METHOD MoveModulo 								: REFERENCE TO Tc2_MC2.ST_McOutputs
VAR_INPUT
	bExecute									: BOOL;
END_VAR
END_METHOD

METHOD MoveModulo2 								: REFERENCE TO Tc2_MC2.ST_McOutputs
VAR_INPUT
	bExecute									: BOOL;
END_VAR
END_METHOD

METHOD MoveModuloClear 							: BOOL
END_METHOD

METHOD MoveModuloClear2 						: BOOL
END_METHOD

METHOD MoveModuloCurrent 						: REFERENCE TO Tc2_MC2.ST_McOutputs
VAR_INPUT
	bExecute									: BOOL;
END_VAR
END_METHOD

METHOD MoveModuloCurrent2 						: REFERENCE TO Tc2_MC2.ST_McOutputs
VAR_INPUT
	bExecute									: BOOL;
END_VAR
END_METHOD

METHOD MoveModuloEx 							: BOOL
END_METHOD

METHOD MoveModuloEx2 							: BOOL
END_METHOD

METHOD MoveModuloNeg 							: REFERENCE TO Tc2_MC2.ST_McOutputs
VAR_INPUT
	bExecute									: BOOL;
END_VAR
END_METHOD

METHOD MoveModuloNeg2 							: REFERENCE TO Tc2_MC2.ST_McOutputs
VAR_INPUT
	bExecute									: BOOL;
END_VAR
END_METHOD

METHOD MoveModuloPos 							: REFERENCE TO Tc2_MC2.ST_McOutputs
VAR_INPUT
	bExecute									: BOOL;
END_VAR
END_METHOD

METHOD MoveModuloPos2 							: REFERENCE TO Tc2_MC2.ST_McOutputs
VAR_INPUT
	bExecute									: BOOL;
END_VAR
END_METHOD

METHOD MoveModuloShort 							: REFERENCE TO Tc2_MC2.ST_McOutputs
VAR_INPUT
	bExecute									: BOOL;
END_VAR
END_METHOD

METHOD MoveModuloShort2 						: REFERENCE TO Tc2_MC2.ST_McOutputs
VAR_INPUT
	bExecute									: BOOL;
END_VAR
END_METHOD

METHOD MoveRelative 							: REFERENCE TO Tc2_MC2.ST_McOutputs
VAR_INPUT
	bExecute									: BOOL;
END_VAR
END_METHOD

METHOD MoveRelative2 							: REFERENCE TO Tc2_MC2.ST_McOutputs
VAR_INPUT
	bExecute									: BOOL;
END_VAR
END_METHOD

METHOD MoveRelativeClear 						: BOOL
END_METHOD

METHOD MoveRelativeClear2 						: BOOL
END_METHOD

METHOD MoveRelativeEx 							: BOOL
END_METHOD

METHOD MoveRelativeEx2 							: BOOL
END_METHOD

METHOD MoveVelocity 							: REFERENCE TO Tc2_MC2.ST_McOutputs
VAR_INPUT
	bExecute									: BOOL;
END_VAR
END_METHOD

METHOD MoveVelocity2 							: REFERENCE TO Tc2_MC2.ST_McOutputs
VAR_INPUT
	bExecute									: BOOL;
END_VAR
END_METHOD

METHOD MoveVelocityClear 						: BOOL
END_METHOD

METHOD MoveVelocityClear2 						: BOOL
END_METHOD

METHOD MoveVelocityEx 							: BOOL
END_METHOD

METHOD MoveVelocityEx2 							: BOOL
END_METHOD

PROPERTY nErrorId 								: UDINT
GET
END_GET
END_PROPERTY

PROPERTY pAbsolute 								: REFERENCE TO Tc2_MC2.ST_McOutputs
GET
END_GET
SET
END_SET
END_PROPERTY

PROPERTY pAbsolute2 							: REFERENCE TO Tc2_MC2.ST_McOutputs
GET
END_GET
SET
END_SET
END_PROPERTY

PROPERTY pEStop 								: REFERENCE TO Tc2_MC2.ST_McOutputs
GET
END_GET
SET
END_SET
END_PROPERTY

PROPERTY pGear 									: REFERENCE TO Tc2_MC2.ST_McOutputs
GET
END_GET
SET
END_SET
END_PROPERTY

PROPERTY pHalt 									: REFERENCE TO Tc2_MC2.ST_McOutputs
GET
END_GET
SET
END_SET
END_PROPERTY

PROPERTY pHome 									: REFERENCE TO Tc2_MC2.ST_McOutputs
GET
END_GET
SET
END_SET
END_PROPERTY

PROPERTY pJog 									: REFERENCE TO Tc2_MC2.ST_McOutputs
GET
END_GET
SET
END_SET
END_PROPERTY

PROPERTY pLimitSwitch 							: REFERENCE TO Tc2_MC2.ST_McOutputs
GET
END_GET
SET
END_SET
END_PROPERTY

PROPERTY pModulo 								: REFERENCE TO Tc2_MC2.ST_McOutputs
GET
END_GET
SET
END_SET
END_PROPERTY

PROPERTY pModulo2 								: REFERENCE TO Tc2_MC2.ST_McOutputs
GET
END_GET
SET
END_SET
END_PROPERTY

PROPERTY pOut 									: REFERENCE TO Tc2_MC2.ST_McOutputs
GET
END_GET
SET
END_SET
END_PROPERTY

METHOD Power 									: REFERENCE TO Tc2_MC2.ST_McOutputs
END_METHOD

PROPERTY pPower 								: REFERENCE TO Tc2_MC2.ST_McOutputs
GET
END_GET
SET
END_SET
END_PROPERTY

PROPERTY pRelative 								: REFERENCE TO Tc2_MC2.ST_McOutputs
GET
END_GET
SET
END_SET
END_PROPERTY

PROPERTY pRelative2 							: REFERENCE TO Tc2_MC2.ST_McOutputs
GET
END_GET
SET
END_SET
END_PROPERTY

PROPERTY pReset 								: REFERENCE TO Tc2_MC2.ST_McOutputs
GET
END_GET
SET
END_SET
END_PROPERTY

PROPERTY pSetPos 								: REFERENCE TO Tc2_MC2.ST_McOutputs
GET
END_GET
SET
END_SET
END_PROPERTY

PROPERTY pStop 									: REFERENCE TO Tc2_MC2.ST_McOutputs
GET
END_GET
SET
END_SET
END_PROPERTY

PROPERTY pVelocity 								: REFERENCE TO Tc2_MC2.ST_McOutputs
GET
END_GET
SET
END_SET
END_PROPERTY

PROPERTY pVelocity2 							: REFERENCE TO Tc2_MC2.ST_McOutputs
GET
END_GET
SET
END_SET
END_PROPERTY

METHOD Reset 									: REFERENCE TO Tc2_MC2.ST_McOutputs
VAR_INPUT
	bExecute									: BOOL;
END_VAR
END_METHOD

METHOD ResetClear 								: BOOL
END_METHOD

METHOD ResetEx 									: BOOL
END_METHOD

METHOD SetPos 									: REFERENCE TO Tc2_MC2.ST_McOutputs
VAR_INPUT
	bExecute									: BOOL;
	bMode										: BOOL;	// RELATIVE=True, ABSOLUTE=False (Default)
	stOptions									: ST_SetPositionOptions;
END_VAR
END_METHOD

METHOD SetPosClear 								: BOOL
END_METHOD

METHOD SetPosEx 								: BOOL
VAR_INPUT
	bMode										: BOOL;	// RELATIVE=True, ABSOLUTE=False (Default)
	stOptions									: ST_SetPositionOptions;
END_VAR
END_METHOD

METHOD Stop 									: REFERENCE TO Tc2_MC2.ST_McOutputs
VAR_INPUT
	bExecute									: BOOL;
END_VAR
END_METHOD

METHOD StopClear 								: BOOL
END_METHOD

METHOD StopEx 									: BOOL
END_METHOD

END_INTERFACE

// ---- POUs/MAIN.TcPOU
PROGRAM MAIN
VAR_INPUT
	bWeighingFormDone											: BOOL;
	IbTwoPhasesFormSensorBetweenDispencers			AT %I*		: BOOL;		// Wejście czujnika pomiedzy dozownikami do przesuwania formatek
	IbFormCheckFormSensor 							AT %I*		: BOOL;		// Wejście wykrycia formatek przed szlabanem
	IbBottleInFormCheckBottleSensor 				AT %I*		: BOOL;		// Wejscie wykrycia butelki przed szlabane
	IbFourthFormCheckFormSensor						AT %I*		: BOOL;	
	IbSecondFormCheckFormSensor						AT %I*		: BOOL;	

	(*CapSorterDrag*)
	IbCapSorterFourthFormCheckFormSensor						: BOOL;
	IbCapSorterBeforeFourthFormCheckFormSensor					: BOOL;
	IbCapSorterAfterFormSensor 									: BOOL;
	IbCapSorterAfterFormSensor2 								: BOOL;		
	IbCapSorterAfterFormSensor3 					AT %I*		: BOOL;			
	IbCapSorterFirstFormCheckFormSensor 						: BOOL;		
	IbLidSealerFirstFormSensor						AT %I*:BOOL;			// Czujnik obecności 2-ej formatki przygrzewacze platynek
	IbLidSealerSecondFormSensor 								: BOOL;		// Czujnik obecności 2-ej formatki przygrzewacze platynek
	IbLidSealerAfterSensor 										: BOOL;		// Czujnik obecności formatek przygrzewacze platynek wyjazd
	IbBlowBeforeGripperScrewerSensor							: BOOL;
	IbLidFeederThirdFormSensor 							AT %I*  : BOOL;		// Czujnik obecności formatki trzecia formatka 
	IbLidFeederAfterSensor 								AT %I*  : BOOL;		// Czujnik obecności formatki wyjazd	
END_VAR
VAR
	fbReasonBadPackage1											: FB_ReasonBadPackage;
	fbReasonBadPackage2											: FB_ReasonBadPackage;
	fb2ReasonBadPackageWithID									: FB_2ReasonBadPackageWithID;	
	
	fbMRBottleFeederPackageState								: FB_MoveRegister;
	fbMRBeforeDispencersPackageStateNew							: FB_MoveRegister;
	fbMRDispencerPackageState									: FB_MoveRegister4;//Sprzed dozowników na dozowniki
	fbMRAfterDispencerPackageState								: FB_MoveRegister4;//z dozowników za dozowniki
	fbMRWeightPackageState										: FB_MoveRegister; // zza dozowników na wage
	fbMRWeight2PhasePackageState								: FB_MoveRegister; // zza dozowników na wage 2 fazy
	fbMRAfterWeightPackageState									: FB_MoveRegister; // z wagi na transporter
	fbMRBEforeScrewer2PackageState								: FB_MoveRegisterSortAndMove;
	fbMRBeforeScrewerPackageState								: FB_MoveRegisterCapControl; // Przed zakręcarkami

	fbMRCorrectCapPackageState									: FB_MoveRegister; // zza zakręcarek na kontrole zakreceniea
	
// Dodatkowe przesuwanie rejestrów 
	
	fbMRBeforeDispencer34PackageState							: FB_MoveRegister;
	fbMRAfterDispencer34PackageState							: FB_MoveRegister4;
	fbMRDispencer34PackageState									: FB_MoveRegister4;
	fbMRBetweenDispencerPackageState							: FB_MoveRegister; 
	fbMRAfterDispencer12PackageState							: FB_MoveRegister4;
	fbMRDispencer12PackageState									: FB_MoveRegister4;

	
	
// LidFeeder
	fbMRBeforeLidFeeder2PackageState							: FB_MoveRegisterSortAndMoveLF;
	fbMRAfterWeightPackageStateLF								: FB_MoveRegisterLF; // z wagi na transporter
	fbIbLidFeederThirdFormSensor								: FB_InputFilter_V2;
	ftfbIbLidFeederThirdFormSensor								: F_TRIG;
	bMRBeforeLidFeeder2Block									: BOOL;
	rtfbIbLidFeederThirdFormSensor								: R_TRIG;
	ftbMRBeforeLidFeeder2Block									: F_TRIG;
	tofftbMRBeforeLidFeeder2Block								: TOF;	
	bMRLidFeederFormInCap										: BOOL;
// LidFeederDrag
	rtfbLidFeederDrag											: R_TRIG;

//AfterLidFeeder
	fbMRAfterLidFeederPackageState								: FB_MoveRegister; // zza zakręcarek na kontrole zakreceniea
	ftfbIbLidFeederAfterSensor									: F_TRIG;
	rtfbIbLidFeederAfterSensor									: R_TRIG;
	fbIbLidFeederAfterSensor									: FB_InputFilter;

//LidSealer
	rtfbLidSealerDrag											: R_TRIG;
	
	
	fbIbFirstFormCheckFormSensor								: FB_InputFilter_v2;
	fbIbSecondFormCheckFormSensor								: FB_InputFilter_v2;
	fbFilteredFormsSensorGate 									: FB_InputFilter;
	fbIbCapCorrectCheckFormSensor								: FB_InputFilter;
	fbIbScrewerThirdFormCheckFormSensor							: FB_InputFilter;
	fbIbCapPuttedCheckFormSensor								: FB_InputFilter;
	fbIbCapPuttedCheckFormSensorv2								: FB_InputFilter_v2;
	fbIbWeight1FormSensor										: FB_InputFilter_v2;
	fbIbWeight4FormSensor										: FB_InputFilter_v2;
	fbIbCapPuttedCheckFormSensorAfterStart						: FB_InputFilter;
	fbIbScrewerThirdFormCheckFormSensorAfterStart				: FB_InputFilter;
	
	fbIbBottleFeederFormPresent									: FB_InputFilter;
	
	
	
	
	bRFIDArrayClear												: BOOL;
	bDeletebBottleTransferedToExit								: BOOL;
	bNewRFIDSaved												: BOOL;
	
	bWeighingFormDoneDialog										: BOOL;
	bWeighingFormReset											: BOOL;

	bNewRFIDSaved1												: BOOL;
	bNewRFIDSaved2												: BOOL;
	bNewRFIDSaved3												: BOOL;
	bNewRFIDSaved4												: BOOL;
	//Sygnały obecnosci formatek przed dozownikami

	
	
	
	bKeepTryingMove1,bKeepTryingMove2,bKeepTryingMove3,bKeepTryingMove4  		: BOOL;
	bKeepTryingMove5,bKeepTryingMove6,bKeepTryingMove7,bKeepTryingMove8	 		: BOOL;
	bKeepTryingMove9,bKeepTryingMove10,bKeepTryingMove11,bKeepTryingMove12	 	: BOOL;
	bKeepTryingMove13,bKeepTryingMove14,bKeepTryingMove15	 					: BOOL;
	bKeepTryingMove17,bKeepTryingMove18,bKeepTryingMove19,bKeepTryingMove20	 	: BOOL;
	bKeepTryingMove799,bKeepTryingMove798,bKeepTryingMove797,bKeepTryingMove796	 : BOOL;
	
	
	bMRFormExitGate1											: BOOL;
	bMRFormDispencer											: BOOL;
	bMRFormExitDispencer										: BOOL;
	bMRFormExitWeight											: BOOL;
	bMRFormInCap												: BOOL;
	bMRCapCorrect												: BOOL;
// Dodatkowe zmienne dla dwufazy
	bMRFormDispencer12											: BOOL;
	bMRFormDispencer34											: BOOL;
	bMRFormExitDispencer12										: BOOL;
	bMRFormExitDispencer34										: BOOL;
	bMRFormBetweenDispencer										: BOOL;
	

	bResetHistory												: BOOL;
	bSimulationForLoop											: BOOL;
	bTestBrakePoint												: BOOL;
	bMRBeforeScrewer2Block										: BOOL;
	bTemp														: BOOL;
	bTrendIbThirdFormCheckFormSensor							: BOOL;
	bTrendFilteredIbThirdFormCheckFormSensor					: BOOL;

	bRFIDSBeforeScrewerWriteToRegister							: BOOL;
	
	
	nFormCounter												: INT;
	nCheckRobotDone												: INT;
	is															: INT;
	iCountSimulation											: INT;
	ir1															: INT;
	ir2															: INT;
	ir3															: INT;
	ir4															: INT;
	ir5															: INT;
	id															: INT;
	ia															: INT;
	iw															: INT;
	iftfbIbCapPuttedCheckFormSensor								: INT;
	iBadPackage1ReasonCount1									: INT;
	iBadPackage1ReasonCount2									: INT;
	iBadPackage1ReasonCount3									: INT;
	iBadPackage2ReasonCount1									: INT;
	iBadPackage2ReasonCount2									: INT;
	iBadPackage2ReasonCount3									: INT;
	ifbIbCapPuttedCheckFormSensorAfterStart						: INT;
	ifbIbScrewerThirdFormCheckFormSensorAfterStart				: INT;
	irtTimerRFIDScrewersWarning									: INT;
	iRFIDSBeforeScrewerWriteToRegister							: INT;
	
	i															: UINT;
	nr1															: UINT;
	nr2															: UINT;
	nr3															: UINT;
	nr4															: UINT;
	nr5															: UINT;	
	nr6															: UINT;	
	nr7															: UINT;	
	nr8															: UINT;	
	
	nSimulationCardNumber										: ULINT;

	sBadPackage1Reason1											: STRING;
	sBadPackage1Reason2											: STRING;
	sBadPackage1Reason3											: STRING;
	sBadPackage2Reason1											: STRING;
	sBadPackage2Reason2											: STRING;
	sBadPackage2Reason3											: STRING;
	
	// RFID
	rtReadedCardDispencer										: R_TRIG;
	rtReadedCardBeforeScrewers									: R_TRIG;
	rtReadedCardAfterScrewers									: R_TRIG;	
	rtReadedCardAfterDispencers									: R_TRIG;
	rtReadedCardAfterDispencers2Phase							: R_TRIG;
	rtReadedCardLidFeeder										: R_TRIG;
	rtReadedCardLidSealer										: R_TRIG;
	rtReadedCardCapSorter										: R_TRIG;	
	rtReadedCardRobotTransfer									: R_TRIG;
	fbrtReadedCardRobotTransfer									: FB_InputFilter_v2;
	fbrtReadedCardAfterScrewers									: FB_InputFilter_v2;
	rtWeighingForm												: R_TRIG;
	rtWeightingDone												: R_TRIG;
	rtBeforeGateDispencerStateNotPresent						: R_TRIG;
	rtBeforeGateDispencerFormPresent							: R_TRIG;
	rtSimulationSetRegisters									: R_TRIG;
	ftfbIbFirstFormCheckFormSensor								: F_TRIG;
	rtfbIbFirstFormCheckFormSensor								: R_TRIG;

	rtfbIbSecondFormCheckFormSensor								: R_TRIG;
	ftfbIbSecondFormCheckFormSensor								: F_TRIG;
	ftfbIbCapCorrectCheckFormSensor								: F_TRIG;
	rtfbIbCapCorrectCheckFormSensor								: R_TRIG;	
	rtfbFormsDragingPneumaticStationDragging					: R_TRIG;
	ftfbIbScrewerThirdFormCheckFormSensor						: F_TRIG;
	ftfbIbCapPuttedCheckFormSensor								: F_TRIG;
	ftfbIbWeight1FormSensor										: F_TRIG;
	ftIbWeight4FormSensor										: F_TRIG;
	ftbMRBeforeScrewer2Block									: F_TRIG;
	rttonDelayAfterStart										: R_TRIG;
	rtfbIbScrewerThirdFormCheckFormSensor						: R_TRIG;
	rtTimerRFIDScrewersWarning									: R_TRIG;
	
	diRFIDWeightingFormNumber									:DINT;
	tonAfter1stweight											:TON;
	bWeightEnd													:BOOL;
	
	tonWeighingForm												: TON;
	tonFourthFormBeforeDispencerCheck							: TON;
	tofCycleExecute												: TOF;
	tonFormBeforeDispenscerCheck								: TON;
	tonDispencerRepair1											: TON;
	TimerRFIDWeightWarning										: TON;
	tonRobotPackageStatebBottleTransferedToLabeler				: TON;
	tonRobotPackageStatebBottleTransferedToLabeler2				: TON;
	TimerRFIDDispencersWarning									: TON;
	TimerRFIDDispencers2PhaseWarning							: TON;
	TimerRFIDScrewersWarning									: TON;
	TimerRFIDRobotWarning										: TON;
	tofftbMRBeforeScrewer2Block									: TOF;
	tonAfterDispencersRepair									: TON;
	tonAfterDispencersRepair1B									: TON;
	tonAfterDispencersRepair2									: TON;	
	tonAfterDispencersRepair3									: TON;	
	tonAfterDispencersRepair4									: TON;	
	tonRepairLidFeeder1											: TON;		
	tonRepairLidFeeder2											: TON;	
	tonRepairLidFeeder3											: TON;	
	tonRepairLidFeeder4											: TON;	
		
	// dodatkowe zmienne przy dwufazie
	fbIbWeight5FormSensor										: FB_InputFilter_v2;
	fbIbWeight6FormSensor										: FB_InputFilter_v2;

	ftfbIbWeight5FormSensor										: F_TRIG;
	ftIbWeight6FormSensor										: F_TRIG;
	
	//
	
	
	
	rtWeightingDone2Phase										: R_TRIG;
	ftfbIbBottleFeederFormPresent								: F_TRIG;
	
	rtibBottleFeederrFormPresent									: R_TRIG;
	bBitTestOn: BOOL;
	tonFormBeforeDispenscer2PhaseCheck							: TON;
	bTestCounterDispencer										: INT;
	tonRobotPackageStateFormsTooLong							: TON;
	tonRobotPackageState1FormsTooLong							: TON;
	tonRobotPackageState2FormsTooLong							: TON;
	END															: INT;
	ftFormSensorBetweenDispencer								: F_TRIG;
	
	fbIbFormSensorBetweenDispencer								: FB_InputFilter_v2;
	
	tonUnderScrewerFormStuck1									: TON;
	tonUnderScrewerFormStuck2									: TON;
	tonAfterScrewerFormStuck1									: TON;
	iRFIDClearNr1AfterRobotCount								: INT;
	iRFIDClearNr2AfterRobotCount								: INT;
	rtiBottleTransferCase2										: R_TRIG;
	tonAfterDispencer12Repair									: TON;
	rttonAfterDispencer12Repair									: R_TRIG;
	
	tonAfterDispencer1234Repair									: TON;
	tonAfterDispencer1234Repair2								: TON;
	
	tonWeightRepair1											: TON;
	tonWeightRepair2											: TON;	
	rttonAfterDispencer1234Repair								: R_TRIG;
	tonFourhtFormBeforeDispencer34								: TON;
	rttonFourtFormBeforeDispencer34Repair						: R_TRIG;
	rtFormSensorBetweenDispencer								: R_TRIG;
	fbIbCapCorrectCheckAfterScrewerFormSensor					: FB_InputFilter;
	ftfbIbCapCorrectCheckAfterScrewerFormSensor					: F_TRIG;
	
	rtTimerRFIDDispencerWarning: R_TRIG;
	irtTimerRFIDDispencerWarning: INT;
	tWeightTime: TIME;
	
	(*RFID*)
	bRFIDRepairAddNumber								: BOOL;
	iRFIDRepairAddNumber								: INT;
	nRFIDRepairOrderFirstNumber							: ULINT;
	AbRFIDRepairOrderTemp								: ULINT;
	nRFIDRepairToRotate									: ULINT;
	nRFIDRepairFormToRotateCount						: ULINT;
	bRFIDRepairChanged									: BOOL;
	iWeightPackageState12nCardNumberChangeCounter		: INT;
	iWeightPackageState13nCardNumberChangeCounter		: INT;


	
	bRFIDRepairReset: BOOL;
	rtRFIDRepairAddNumber: R_TRIG;
	nBeforeGatePackageState1nCardNumber: ULINT;
	ftRFIDRepairAddNumber: F_TRIG;
	rtRFIDRepairToRotate: R_TRIG;
	nRFIDRepairToRotateBefore: ULINT;
	fbRFIDRepairFilteredFormsSensorGate: FB_InputFilter;
	iRFIDRepairCount1: INT;
	iRFIDRepairCount2: INT;
	iRFIDRepairCount3: INT;
	iRFIDRepairCount4: INT;
	iRFIDRepairCount5: INT;
	bRFIDRepairOrderFirstNumberSaved: BOOL;
	iRFIDRepairCount6: INT;
	iRFIDRepairCount7: INT;
	iWeightPackageState43nCardNumberChangeCounter: INT;
	iWeightPackageState41nCardNumberChangeCounter: INT;
	iWeightPackageState21nCardNumberChangeCounter: INT;
	iWeightPackageState32nCardNumberChangeCounter: INT;
	iWeightPackageState31nCardNumberChangeCounter: INT;
	iUnderScrewerPackageState21nCardNumberChangeCounter: INT;
	iRFIDRepairCount8: INT;
	iRFIDRepairNumberOfForms: INT;
	iUnderScrewerPackageState12nCardNumberChangeCounter: INT;

	rtbBottleDragingStationRun: R_TRIG;
	rtDispencerDragStation: R_TRIG;

	rttonUnderScrewerFormStuck1: R_TRIG;
	rttonRobotPackageStatebBottleTransferedToLabeler: R_TRIG;
	rttonRobotPackageStatebBottleTransferedToLabeler2: R_TRIG;
	rttonRobotPackageState1FormsTooLong: R_TRIG;
	rttonRobotPackageState2FormsTooLong: R_TRIG;
	rteUnderScrewerPackageStateCheck: R_TRIG;
	rteUnderScrewerPackageStateCheck2: R_TRIG;
	iUnderScrewerPackageStateCheckCounter: INT;
	iUnderScrewerPackageStateCheckCounter2: INT;
	tonDispencer34DosingAborted: TON;
	rttonDispencer34DosingAborted: R_TRIG;
	
	tonFormatSensorOn	:	ton;
	tonFormatSensorOff	:	ton;
	bFormatSensor		:	BOOL;

	tonBottleSensorOn	:	ton;
	tonBottleSensorOff	:	ton;
	bBottleSensor		:	BOOL;
	

	
	
	tonIbCapSorterAfterFormSensor						: TON;
	fbMRAfterCapSorterPackageState						: FB_MoveRegister4; // Z sortera za sorter
	fbMRCapSorterPackageState							: FB_MoveRegister4; // Sprzed sortera na sorter
	fbMRBeforeCapSorterPackageState						: FB_MoveRegister;
	fbFilteredCapSorterFormsSensorGate 					: FB_InputFilter;
	ftfbFilteredCapSorterFormsSensorGate				: F_TRIG;
	tonFormBeforeCapSorterCheck							: TON;
	
	
	iAfterDispencersFormCounter: INT;
	itonFormBeforeCapSorterCheck: INT;
	bResetAntyErrorCounters: BOOL;
	lrAnRFIDWeightShowAverage: LREAL;
	iAnRFIDWeightShowAverageCount: INT;
	bRFIDWeightShowAverageError: BOOL;	
	ii: UINT;
	

	
	iLFTest1: INT;
	j: INT;
	iTestCCC1: INT;
	iTestCCC2: INT;
	
	(*ROPP*)
	rtReadedCardBeforeROPP				: R_TRIG;
	rtReadedCardAfterROPP				: R_TRIG;
	iropp1, iropp2						: INT;
	bRFIDSBeforeROPPWriteToRegister		: BOOL;
	iRFIDSBeforeROPPWriteToRegister		: INT;
	rtfbROPPDrag						: R_TRIG;
	bMRBeforeROPP2Block					: BOOL;
	ftbMRBeforeROPP2Block 				: F_TRIG;
	tofftbMRBeforeROPP2Block			: TOF;
	fbMRBEforeROPP2PackageState			: FB_MoveRegisterSortAndMoveROPP;
	bKeepTryingMoveROPP1					: BOOL;	
	bROPPMR								: BOOL;	
	fbMRBeforeROPPPackageState			: FB_MoveRegisterROPPCapControl; 
	tonRepairROPP1						: TON;		
	tonRepairROPP2						: TON;	
	tonRepairROPP3						: TON;	
	tonRepairROPP4						: TON;		
	bKeepTryingMoveROPP2				: BOOL;
	iPodglad:UINT;
	
	fbShutdown_UBL :NT_Shutdown;
	fbShutdown_UCF :NT_Shutdown;
	fbShutdown_UBF :NT_Shutdown;
	
	 fbRenew : FB_AutoTrialRenew_ADS;
     bExpired : BOOL := FALSE;
	 btestlicense	:bool:=false;
END_VAR

TcMcGlobal.NCPORT_TCMC_RESET := 501; // Przeciw bluescreen'om

VIS.sType				:=	'UL50-0125';
VIS.sSerialNumber		:=	'UL50-0125';
VIS.rProgramVersion		:=	0.2; (*XD*)
VIS.rLastTimeChanges	:=	20252810;


//Resetowanie przeważania
IF bWeighingFormReset THEN
	
	FOR i := 1 TO 100 DO
		VIS.AnRFIDCardNumberShow[i]								:= 0;
		VIS.AnRFIDWeightShow[i]									:= 0;
	END_FOR
	
	bWeighingFormReset 											:= FALSE;
	bWeighingFormDone 											:= FALSE;
	bWeighingFormDoneDialog 									:= FALSE;
	iRFIDRepairCount1	:=0;
	iRFIDRepairCount2	:=0;
	iRFIDRepairCount3	:=0;
	iRFIDRepairCount4	:=0;
END_IF

aInFormatSensorFilter();

aWizard();
P00_SystemDiagnostics();
a0RemoteControl();
aAntyError();
aAntyErrorLidFeeder();
//aAntyErrorROPP();
aBadPackage();
aCycleLogicHMI();
aStatistics();
aSimulation();

//aRFIDRepairSignals();
//MAIN.aRFIDRepairReset();
//bRFIDChecker:=TRUE; 
bRFIDChecker:=FALSE;

IF bRFIDChecker	THEN
	MAIN.aRFIDRepairOrderCreate();
	MAIN.aRFIDRepairOrderSearch();
	MAIN.aRFIDRepairStatistic();
END_IF	

P00_Communication();
P00_PackML();			
P00_Alarms();
P00_Basic();
P00_Counters();
P00_Persistent();
P00_OEE();
P00_PneumaticValves();
P00_ReadRFIDCard();
P00_Recipes();
P00_Signalization();
P00_Visualization();
P01_TwoPhasesBarriers();
P01_BottleFeeder();
P01_PucksInserter();
P01_BottleSorter();
P01_Gates();
P02_BottlePusher();
P02_Dispencers();
P02_DispencersCharts();
P05_WeightCorrection();
//P05_Weight();
P06_LidFeeder();
//P06_WickFeeder();
P06_LidPuttedCheck();
P07_CapPusher();
P06_LidSealer();
P07_ROPP();
P08_CapFeeder();
P08_CapSorter();
P09_CapPuttedCheck();
P10_GripperScrewer();
P11_CapCorrectCheck();
P11_RollerScrewer();
P13_BottleTransfer();
P13_BottleTransferAfterDrag();
P14_BadBottleConyevor();
P15_FormTransporters();
P16_LabelMachine();
P17_TurnTables();
P20_ExhaustFan();
//P030_Recipes();
P010_AlarmsWarningsInfosLogs();
P020_RtcEffectivityOEE();
P009_ReadSavePersistent();
P_AdsLicenseServer();
P200_CapPreScrewer();

tofCycleExecute(IN:=	(P00_PackML.fbPMLAuto.ePMLState = E_PMLState.ePMLState_STARTING) OR (P00_PackML.fbPMLAuto.ePMLState = E_PMLState.ePMLState_EXECUTE) OR 
						(P00_PackML.fbPMLAuto.ePMLState = E_PMLState.ePMLState_STOPPING) OR (P00_PackML.fbPMLAuto.ePMLState = E_PMLState.ePMLState_ABORTING),PT:=T#2S);

IF  tofCycleExecute.Q THEN
	
	IF bDosingTwoPhases THEN
		MAIN.aCycleRegister2Phase();
	ELSE
		IF bLidFeederEnable OR bWickFeederEnable THEN
			MAIN.aCycleRegister1PhaseLidFeederOrWick();
		ELSE
			MAIN.aCycleRegister1Phase();
		END_IF
	END_IF
	
END_IF

aRFIDWarnings();


fbShutdown_UBL(
	NETID:= '192.168.40.180.1.1',
	DELAY:= 10,
	START:=vis.bOffPLC ,
	TMOUT:= ,
	BUSY=> ,
	ERR=> ,
	ERRID=> );
	
//fbShutdown_UCF(
//	NETID:= '192.168.40.155.1.1',
//	DELAY:= 10,
//	START:=vis.bOffPLC ,
//	TMOUT:= ,
//	BUSY=> ,
//	ERR=> ,
//	ERRID=> );	
//	
//fbShutdown_UBF(
//	NETID:= '192.168.40.151.1.1',
//	DELAY:= 10,
//	START:=vis.bOffPLC ,
//	TMOUT:= ,
//	BUSY=> ,
//	ERR=> ,
//	ERRID=> );

IF btestlicense THEN
    bExpired := TRUE;
END_IF
fbRenew(
    bExpired := bExpired,
    sProductId := 'TC1220',
    sAdsServerNetId := '192.168.40.180.1.1',    // AMS Net ID PLC z serwerem ADS
    nAdsServerPort := 851
);

// Nowa "licencja"
fbRenew.sLicenseOut;

ACTION a0RemoteControl:
(*
Nazwa:			a0RemoteControl
Opis:			Ulatwienie obsługi maszyny bez wizki
Wersja:			v0.1
Data:			2023-03-13
Autor:			DP
Urzadzenia:		
Konfiguracja:	
Info:
-


*)
{warning 'Dorobić błędy Undervoltage'}
VIS.bChooseRecipe ; P00_PackML.iChooseRecipe;
VIS.bRecipeLoading;P00_PackML.fbbRecipeLoading.bOut;

IbCycleStopButton;
IbCycleStartButton; 

VIS.bServiceMode;
VIS.bAllowStart ;
VIS.bSimulation;
VIS.bWeighingForm;

VIS.lrDispencersLifterReadyPositionShow;
VIS.lrDispencer1LifterStartDosePositionShow;
VIS.lrDispencer1LifterStopDosePositionShow;

VIS.bBottleTransferAllFormsToLabeler;
VIS.bBottleTransferAllFormsToExit;
VIS.iBottleTransferSpeedShow;	

stBottleSorterRead.ePackMLMode;
stBottleSorterRead.ePackMLAutoState; 
bBottleSorterDisable;

stCapSorterRead.ePackMLMode;
stCapSorterRead.ePackMLAutoState; 
bCapSorterDisable;
VIS.bCapPuttedCheckIgnoreErrors;

VIS.bResetErrorVisuCmd;
VIS.bErrorOccure;							
VIS.sStationInError;	
VIS.udiStationInError;			
VIS.udiStationErrorCode;			
VIS.sStationErrorDescription;	
VIS.sStationErrorDescription2;	

bHomingDialog;
VIS.bDialogBoxText;
VIS.bDialogBoxAck;

VIS.lrDispencer1DoseVolumeCV					;				// Doza 1 [ml]
VIS.lrDispencer2DoseVolumeCV					;				// Doza 2 [ml]
VIS.lrDispencer3DoseVolumeCV					;				// Doza 3 [ml]	
VIS.lrDispencer4DoseVolumeCV					;				// Doza 4 [ml]	
VIS.lrDispencer1WeightMeasured					;				// Waga z dozownika 1 [g]	
VIS.lrDispencer2WeightMeasured					;				// Waga z dozownika 2 [g]		
VIS.lrDispencer3WeightMeasured					;				// Waga z dozownika 3 [g]	
VIS.lrDispencer4WeightMeasured					;				// Waga z dozownika 4 [g]	
VIS.bDispencer1WeightMeasured					;				// [H] Waga zmierzona z dozownika nr 1	
VIS.bDispencer2WeightMeasured					;				// [H] Waga zmierzona z dozownika nr 2
VIS.bDispencer3WeightMeasured					;				// [H] Waga zmierzona z dozownika nr 3
VIS.bDispencer4WeightMeasured					;				// [H] Waga zmierzona z dozownika nr 4



iRepairFourthFormBeforeDispencerCounter;	// 1A - Ustawianie 4 formatki(*****************Autonaprawa przed dozownikami	*****************)
iRepairBeforeDispencer34Counter;			// 1B (2faza) - Autonaprawa 2 formatki przed dozowikiem 34
iCounterDispencer34DosingAborted;			// 1C (2faza) - Autonaprawa jak jest butelka a niewydozowało
iRepairFormBeforeDispenscerCounter;			// 1D - Ustawianie jak nie ma dwufazy - Ustawianie 1 2 3 4 formatki
iRepairFormBeforeDispenscer2PhaseCounter;	// 1E (2faza) - ustawianie jak jest dwufaza - Ustawianie 1 2  formatki
itonAfterDispencersRepair;					// 1 - Kasowanie rejestrow jezeli nie ma nic na czujnikach (******************Autonaprawa za dozownikami*************************)
itonAfterDispencersRepair2;					// 2 - Kasowanie rejestrow jezeli nei ma nic na czujnikach----------------
itonAfterDispencersRepair3;					// 3 - Kasowanie rejestrow jezeli nei ma nic na czujnikach --------------
itonAfterDispencersRepair4;					// 4 -  Kasowanie rejestrow jezeli nei ma nic na czujnikach-------------
iRepairAfterDispencerCounter;				// 4 - Kssowanie za 1 i 2 dozownikiem jak dwufaza -----------------------
iRepairBeforeDispencer12Counter;			// 5 - Dodawanie formatek przed 12 jak stoją za 34 ---------------------
iRepairBeforeDispencer12Counter2;
itonFormBeforeCapSorterCheck;				// 1A - Ustawianie 1 2 3 4 formatki(*****Autonaprawa pod sorterem nasadek**********)
iScrewerFormStuck;							// 1A - (****** Autonaprawa pod zakręcarkami*********)
iScrewerFormStuck2;							// 1B - jezeli nie odczyta przed zakrecarkami
iScrewerFormStuck3;							// 1S - jezeli nie ma za zakrecarka
iRobotRepairPackageForm1Counter;			// Jak jest przeniesiona na etykieciarke(*****Autonaprawa pod robotem**********)
iRobotRepairPackageForm2Counter;
itonRobotBottleTransferedToLabelerRepair;
itonRobotBottleTransferedToLabeler2Repair;
END_ACTION

ACTION a2RFID:
(*
Nazwa:			aRFID
Opis:			Zapisywanie RFID
Wersja:			v0.5
Data:			2024-12-02
Autor:			DP
Urzadzenia:		
Konfiguracja:	
Zmiany:
Info:
- zapis RFID do struktury
- text
*)

(*********************Wywoływane w aCycleLogic************************)

(*******************************)
(***CZUJNIK PRZED DOZOWNIKAMI***)

//Jeżeli wykryło kartę 
rtReadedCardDispencer(CLK:=P00_ReadRFIDCard.bReadedCardDispencer,Q=>);
IF rtReadedCardDispencer.Q THEN
	nr1:=nr1+1;
	eBeforeGatePackageState[1].bFormPresent:=TRUE; // dodane do testów jak cos to wykomentować 20.06
	IF eBeforeGatePackageState[1].bFormPresent THEN
		eBeforeGatePackageState[1].nCardNumber:=P00_ReadRFIDCard.nReadedCardDispencer;
		
		//Dodawanie RFID do tablicy
		FOR ir1 := 1 TO 100 DO
					 IF eRFID[ir1].nCardNumber = P00_ReadRFIDCard.nReadedCardDispencer THEN
						 	IF NOT nCheckWeiginhForm THEN
								eRFID[ir1] := eClearPackageState;
							END_IF
							eRFID[ir1].nCardNumber := P00_ReadRFIDCard.nReadedCardDispencer;
							eRFID[ir1].bFormPresent := eBeforeGatePackageState[1].bFormPresent;
							eRFID[ir1].bBottlePresent := eBeforeGatePackageState[1].bBottlePresent;
							eRFID[ir1].nID := eBeforeGatePackageState[1].nID;
							bNewRFIDSaved := TRUE;
					 END_IF
		END_FOR	
		//Dodawanie nowego numeru do RFID jeżeli nie jest w tablicy
		IF NOT bNewRFIDSaved THEN
				FOR ir1 := 1 TO 100 DO
					 IF eRFID[ir1].nCardNumber = 0 THEN
							eRFID[ir1] := eClearPackageState;
							eRFID[ir1].nCardNumber := P00_ReadRFIDCard.nReadedCardDispencer;
							eRFID[ir1].bFormPresent := TRUE;					
							eRFID[ir1].bBottlePresent := eBeforeGatePackageState[1].bBottlePresent;
							eRFID[ir1].nID := eBeforeGatePackageState[1].nID;				
							EXIT;
					 END_IF
				END_FOR	
		END_IF
		bNewRFIDSaved := FALSE;	
	ELSE
		bTestBrakePoint;	
	END_IF	
END_IF
(**KONIEC CZUJNIK PRZED DOZOWNIKAMI**)
(************************************)


(**********************************************)
(************CZUJNIK ZA Dozownikami ***********)

//Jeżeli wykryło kartę 
rtReadedCardAfterDispencers(CLK:=P00_ReadRFIDCard.bReadedCardAfterDispencers,Q=>);
IF rtReadedCardAfterDispencers.Q THEN
	eAfterDispencersPackageState[1].bFormPresent := true; // ZMIANA 16032022
	nr2:=nr2+1;
	IF (eAfterDispencersPackageState[1].bFormPresent) AND P00_ReadRFIDCard.nReadedCardAfterDispencers > 0 THEN
		eAfterDispencersPackageState[1].nCardNumber:=P00_ReadRFIDCard.nReadedCardAfterDispencers;		
		FOR ir2 := 1 TO 100 DO
			 IF eRFID[ir2].nCardNumber = P00_ReadRFIDCard.nReadedCardAfterDispencers THEN
					eRFID[ir2].nCardNumber := P00_ReadRFIDCard.nReadedCardAfterDispencers;
					eRFID[ir2].bFormPresent := eAfterDispencersPackageState[1].bFormPresent;	
					eAfterDispencersPackageState[1]:=eRFID[ir2];//Zapisywanie tablicy do wglądu w HMI						
					bNewRFIDSaved := TRUE;
			 END_IF
		END_FOR	
			IF NOT bNewRFIDSaved THEN
				FOR ir2 := 1 TO 100 DO
					 IF eRFID[ir2].nCardNumber = 0 THEN
						eRFID[ir2] := eClearPackageState;
						eRFID[ir2].nCardNumber := P00_ReadRFIDCard.nReadedCardAfterDispencers;
						eRFID[ir2].bFormPresent := TRUE;
						EXIT;
					 END_IF
				END_FOR	
			END_IF
	bNewRFIDSaved := FALSE;	
	END_IF
END_IF

(**********************************************)
(************CZUJNIK ZA Dozownikami 2 faza*****)

//Jeżeli wykryło kartę 
rtReadedCardAfterDispencers2Phase(CLK:=P00_ReadRFIDCard.bReadedCardAfterDispencers2Phase,Q=>);
IF rtReadedCardAfterDispencers2Phase.Q THEN
	eAfterDispencer12PackageState2Phase[1].bFormPresent := TRUE; // ZMIANA 16032022
	nr6:=nr6+1;
	IF (eAfterDispencer12PackageState2Phase[1].bFormPresent) AND P00_ReadRFIDCard.nReadedCardAfterDispencers2Phase > 0 THEN
		eAfterDispencer12PackageState2Phase[1].nCardNumber:=P00_ReadRFIDCard.nReadedCardAfterDispencers2Phase;		
		FOR nr6 := 1 TO 100 DO
			 IF eRFID[nr6].nCardNumber = P00_ReadRFIDCard.nReadedCardAfterDispencers2Phase THEN
					eRFID[nr6].nCardNumber := P00_ReadRFIDCard.nReadedCardAfterDispencers2Phase;
					eRFID[nr6].bFormPresent := eAfterDispencer12PackageState2Phase[1].bFormPresent;	
					eAfterDispencer12PackageState2Phase[1]:=eRFID[nr6];//Zapisywanie tablicy do wglądu w HMI						
					bNewRFIDSaved := TRUE;
			 END_IF
		END_FOR	
			IF NOT bNewRFIDSaved THEN
				FOR nr6 := 1 TO 100 DO
					 IF eRFID[nr6].nCardNumber = 0 THEN
						eRFID[nr6] := eClearPackageState;
						eRFID[nr6].nCardNumber := P00_ReadRFIDCard.nReadedCardAfterDispencers2Phase;
						eRFID[nr6].bFormPresent := TRUE;
						EXIT;
					 END_IF
				END_FOR	
			END_IF
	bNewRFIDSaved := FALSE;	
	END_IF
END_IF

IF NOT P05_Weight.IbWeight6FormSensor AND NOT MAIN.IbSecondFormCheckFormSensor AND VIS.bGateBeforeWeight56Run=FALSE THEN
	eAfterDispencer12PackageState2Phase[1].bFormPresent :=FALSE;
	eAfterDispencer12PackageState2Phase[2].bFormPresent	:=FALSE;
END_IF

(*************************************************)
(*(************CZUJNIK PRZED Nakładaniem PLATYNEK***********)
//Jeżeli wykryło kartę 
rtReadedCardLidFeeder(CLK:=P00_ReadRFIDCard.bReadedCardLidFeeder,Q=>);
IF rtReadedCardLidFeeder.Q THEN
//	eAfterLidFeederPackageState[1].bFormPresent := TRUE; 
	nr8:=nr8+1;
	IF (eAfterLidFeederPackageState[1].bFormPresent) AND P00_ReadRFIDCard.nReadedCardLidFeeder > 0 THEN
		eAfterLidFeederPackageState[1].nCardNumber:=P00_ReadRFIDCard.nReadedCardLidFeeder;		
		FOR nr8 := 1 TO 100 DO
			 IF eRFID[nr8].nCardNumber = P00_ReadRFIDCard.nReadedCardLidFeeder THEN
					eRFID[nr8].nCardNumber := P00_ReadRFIDCard.nReadedCardLidFeeder;
					eRFID[nr8].bFormPresent := eAfterLidFeederPackageState[1].bFormPresent;	
					eAfterLidFeederPackageState[1]:=eRFID[nr8];//Zapisywanie tablicy do wglądu w HMI						
					bNewRFIDSaved := TRUE;
			 END_IF
		END_FOR	
			IF NOT bNewRFIDSaved THEN
				FOR nr8 := 1 TO 100 DO
					 IF eRFID[nr8].nCardNumber = 0 THEN
						eRFID[nr8] := eClearPackageState;
						eRFID[nr8].nCardNumber := P00_ReadRFIDCard.nReadedCardLidFeeder;
						eRFID[nr8].bFormPresent := TRUE;
						EXIT;
					 END_IF
				END_FOR	
			END_IF
	bNewRFIDSaved := FALSE;	
	END_IF
END_IF
//IF P00_PackML.fbIbLidFeederAfterSensorLonger.bOUT THEN
//	eAfterLidFeederPackageState[1].bFormPresent:=FALSE;
//END_IF*)

(*************************************************)
(************CZUJNIK PRZED ZGRZEWANIEM PLATYNEK***********)
//Jeżeli wykryło kartę 
rtReadedCardLidSealer(CLK:=P00_ReadRFIDCard.bReadedCardLidSealer,Q=>);
IF rtReadedCardLidSealer.Q THEN
//	eAfterLidFeederPackageState[1].bFormPresent := TRUE; 
	nr8:=nr8+1;
	IF (eAfterLidFeederPackageState[1].bFormPresent) AND P00_ReadRFIDCard.nReadedCardLidSealer > 0 THEN
		eAfterLidFeederPackageState[1].nCardNumber:=P00_ReadRFIDCard.nReadedCardLidSealer;		
		FOR nr8 := 1 TO 100 DO
			 IF eRFID[nr8].nCardNumber = P00_ReadRFIDCard.nReadedCardLidSealer THEN
					eRFID[nr8].nCardNumber := P00_ReadRFIDCard.nReadedCardLidSealer;
					eRFID[nr8].bFormPresent := eAfterLidFeederPackageState[1].bFormPresent;	
					eAfterLidFeederPackageState[1]:=eRFID[nr8];//Zapisywanie tablicy do wglądu w HMI						
					bNewRFIDSaved := TRUE;
			 END_IF
		END_FOR	
			IF NOT bNewRFIDSaved THEN
				FOR nr8 := 1 TO 100 DO
					 IF eRFID[nr8].nCardNumber = 0 THEN
						eRFID[nr8] := eClearPackageState;
						eRFID[nr8].nCardNumber := P00_ReadRFIDCard.nReadedCardLidSealer;
						eRFID[nr8].bFormPresent := TRUE;
						EXIT;
					 END_IF
				END_FOR	
			END_IF
	bNewRFIDSaved := FALSE;	
	END_IF
END_IF
//IF P00_PackML.fbIbLidFeederAfterSensorLonger.bOUT THEN
//	eAfterLidFeederPackageState[1].bFormPresent:=FALSE;
//END_IF

(*************************************************)
(************CZUJNIK PRZED ROPP***********)
//Jeżeli wykryło kartę 
rtReadedCardBeforeROPP(CLK:=P07_ROPP.bReadedCardBeforeROPP,Q=>);
IF rtReadedCardBeforeROPP.Q THEN
	eBeforeROPPCapControlPackageState[1].bFormPresent := TRUE; 
	IF eBeforeROPPCapControlPackageState[1].bFormPresent THEN
		eBeforeROPPCapControlPackageState[1].nCardNumber:=P07_ROPP.nReadedCardBeforeROPP;		
		FOR iropp1 := 1 TO 100 DO
			 IF eRFID[iropp1].nCardNumber = P07_ROPP.nReadedCardBeforeROPP THEN
				//eRFID[iropp1].nCardNumber		:= P07_ROPP.nReadedCardBeforeROPP;
				eRFID[iropp1].bFormPresent		:= eBeforeROPPCapControlPackageState[1].bFormPresent;
				IF eRFID[iropp1].bBottlePresent THEN
					eBeforeROPPCapControlPackageState[1].bBottlePresent := TRUE;
				END_IF
				IF eRFID[iropp1].bWeightOK THEN
					eBeforeROPPCapControlPackageState[1].bWeightOK := TRUE;
				END_IF				
	           
				(*Dodatkowy kod jeżeli nasadka została sprawdzona wczesniej niż odczytał czujnik RFID*) 	
				eRFID[iropp1].bROPPPutted 		:= eBeforeROPPCapControlPackageState[1].bROPPPutted; 	
				eRFID[iropp1].bROPPPuttedChecked:= eBeforeROPPCapControlPackageState[1].bROPPPuttedChecked; 	
				IF eBeforeROPPCapControlPackageState[1].bROPPPutted THEN					
					eRFID[iropp1].bBottlePresent := TRUE;						
				END_IF	
				(*Koniec Dodatkowy kod jeżeli nasadka została sprawdzona wczesniej niż odczytał czujnik RFID*)
			
				//eBeforeROPPCapControlPackageState[1]	:=	eRFID[iropp1];//Zapisywanie tablicy do wglądu w HMI						
				bNewRFIDSaved							:=	TRUE;
				bRFIDSBeforeROPPWriteToRegister 		:=	TRUE;
				iRFIDSBeforeROPPWriteToRegister 		:=	iRFIDSBeforeROPPWriteToRegister + 1;
			 END_IF
		END_FOR	
			IF NOT bNewRFIDSaved THEN
				FOR iropp1 := 1 TO 100 DO
					 IF eRFID[iropp1].nCardNumber = 0 THEN
						eRFID[iropp1]					:= eClearPackageState;
						eRFID[iropp1].nCardNumber		:= P07_ROPP.nReadedCardBeforeROPP;
						eRFID[iropp1].bFormPresent		:= TRUE;
						bRFIDSBeforeROPPWriteToRegister := TRUE;
						EXIT;
					 END_IF
				END_FOR	
			END_IF
	bNewRFIDSaved := FALSE;	
	END_IF
END_IF

(*************************************************)
(************CZUJNIK ZA ROPP**************)
rtReadedCardAfterROPP(CLK:=P07_ROPP.bReadedCardAfterROPP,Q=>);
IF rtReadedCardAfterROPP.Q THEN
	eUnderROPPCorrectCapPackageState[1].bFormPresent := TRUE; 
	IF eUnderROPPCorrectCapPackageState[1].bFormPresent THEN
		eUnderROPPCorrectCapPackageState[1].nCardNumber		:=	P07_ROPP.nReadedCardAfterROPP;		
		FOR iropp2 := 1 TO 100 DO
			 IF eRFID[iropp2].nCardNumber = P07_ROPP.nReadedCardAfterROPP THEN
					eRFID[iropp2].nCardNumber			:=	P07_ROPP.nReadedCardAfterROPP;	
					bNewRFIDSaved					:=	TRUE;
					EXIT;
			 END_IF
		END_FOR	
		IF NOT bNewRFIDSaved THEN
			FOR iropp2 := 1 TO 100 DO
				 IF eRFID[iropp2].nCardNumber = 0 THEN
					eRFID[iropp2]					:=	eClearPackageState;
					eRFID[iropp2].nCardNumber		:=	P07_ROPP.nReadedCardAfterROPP;
					eRFID[iropp2].bFormPresent 		:=	TRUE;
					EXIT;
				 END_IF
			END_FOR	
		END_IF
		bNewRFIDSaved := FALSE;	
	END_IF	
END_IF


(**********************************************)
(************CZUJNIK Przed sorterem********)

//Jeżeli wykryło kartę 
//rtReadedCardCapSorter(CLK:=P00_ReadRFIDCard.bReadedCardCapSorter,Q=>);
rtReadedCardCapSorter(CLK:=fbFilteredCapSorterFormsSensorGate.bOUT,Q=>);//opózniony o 50ms żeby już był wczytany RFID
IF rtReadedCardCapSorter.Q THEN
	eBeforeGateCapSorterPackageState[1].bFormPresent := TRUE; 
	nr7:=nr7+1;
	IF (eBeforeGateCapSorterPackageState[1].bFormPresent) AND P00_ReadRFIDCard.nReadedCardCapSorter > 0 THEN
		eBeforeGateCapSorterPackageState[1].nCardNumber:=P00_ReadRFIDCard.nReadedCardCapSorter;		
		FOR nr7 := 1 TO 100 DO
			 IF eRFID[nr7].nCardNumber = P00_ReadRFIDCard.nReadedCardCapSorter THEN
					eRFID[nr7].nCardNumber := P00_ReadRFIDCard.nReadedCardCapSorter;
					eRFID[nr7].bFormPresent := eBeforeGateCapSorterPackageState[1].bFormPresent;	
					eBeforeGateCapSorterPackageState[1]:=eRFID[nr7];//Zapisywanie tablicy do wglądu w HMI						
					bNewRFIDSaved := TRUE;
			 END_IF
		END_FOR	
			IF NOT bNewRFIDSaved THEN
				FOR nr7 := 1 TO 100 DO
					 IF eRFID[nr7].nCardNumber = 0 THEN
						eRFID[nr7] := eClearPackageState;
						eRFID[nr7].nCardNumber := P00_ReadRFIDCard.nReadedCardCapSorter;
						eRFID[nr7].bFormPresent := TRUE;
						EXIT;
					 END_IF
				END_FOR	
			END_IF
	bNewRFIDSaved := FALSE;	
	END_IF
END_IF



IF P09_CapPuttedCheck.rtCapPuttedFormCheck.Q THEN
	eBeforeCapControlPackageState[1].bFormPresent:=TRUE;
END_IF

(*************************************************)
(************CZUJNIK PRZED ZAKRĘCARKAMI***********)
//Jeżeli wykryło kartę 
rtReadedCardBeforeScrewers(CLK:=P00_ReadRFIDCard.bReadedCardBeforeScrewer,Q=>);
IF rtReadedCardBeforeScrewers.Q THEN
	nr3:=nr3+1;
	eBeforeCapControlPackageState[1].bFormPresent := TRUE; //ZMIANA UBL50 
	IF eBeforeCapControlPackageState[1].bFormPresent THEN
		eBeforeCapControlPackageState[1].nCardNumber:=P00_ReadRFIDCard.nReadedCardBeforeScrewer;		
		FOR ir3 := 1 TO 100 DO
					 IF eRFID[ir3].nCardNumber = P00_ReadRFIDCard.nReadedCardBeforeScrewer THEN
							eRFID[ir3].nCardNumber := P00_ReadRFIDCard.nReadedCardBeforeScrewer;
							eRFID[ir3].bFormPresent := eBeforeCapControlPackageState[1].bFormPresent;
	
							(*Dodatkowy kod jeżeli nasadka została sprawdzona wczesniej niż odczytał czujnik RFID*)
							eRFID[ir3].bCapOK 		:= eBeforeCapControlPackageState[1].bCapOK;		 	
							eRFID[ir3].bCapPutted 	:= eBeforeCapControlPackageState[1].bCapPutted; 	
							eRFID[ir3].bCapChecked	:= eBeforeCapControlPackageState[1].bCapChecked; 	
							IF eBeforeCapControlPackageState[1].bCapOK THEN					
								eRFID[ir3].bBottlePresent := TRUE;						
							END_IF	
							(*Koniec Dodatkowy kod jeżeli nasadka została sprawdzona wczesniej niż odczytał czujnik RFID*)
						
							eBeforeCapControlPackageState[1]:=eRFID[ir3];//Zapisywanie tablicy do wglądu w HMI						
							bNewRFIDSaved:= TRUE;
							bRFIDSBeforeScrewerWriteToRegister := TRUE;
							iRFIDSBeforeScrewerWriteToRegister := iRFIDSBeforeScrewerWriteToRegister + 1;
					 END_IF
		END_FOR	
			IF NOT bNewRFIDSaved THEN
				FOR ir3 := 1 TO 100 DO
					 IF eRFID[ir3].nCardNumber = 0 THEN
							eRFID[ir3] := eClearPackageState;
							eRFID[ir3].nCardNumber := P00_ReadRFIDCard.nReadedCardBeforeScrewer;
							eRFID[ir3].bFormPresent := TRUE;
							bRFIDSBeforeScrewerWriteToRegister := TRUE;
							EXIT;
					 END_IF
				END_FOR	
			END_IF
	bNewRFIDSaved := FALSE;	
	END_IF
END_IF


(*************************************************)
(************CZUJNIK ZA ZAKRĘCARKAMI**************)
fbrtReadedCardAfterScrewers(bIn:=P00_ReadRFIDCard.bReadedCardAfterScrewer,	tFilterTimeOn:=T#10MS,	tFilterTimeOff:=T#0MS);	//opózniony o 50ms żeby już był wczytany RFID
rtReadedCardAfterScrewers(CLK:=fbrtReadedCardAfterScrewers.bOUT,Q=>);
IF rtReadedCardAfterScrewers.Q THEN
	nr4:=nr4+1;
	eUnderCorrectCapPackageState[1].bFormPresent := TRUE; 
	IF eUnderCorrectCapPackageState[1].bFormPresent THEN
		eUnderCorrectCapPackageState[1].nCardNumber		:=	P00_ReadRFIDCard.nReadedCardAfterScrewer;		
		FOR ir4 := 1 TO 100 DO
			 IF eRFID[ir4].nCardNumber = P00_ReadRFIDCard.nReadedCardAfterScrewer THEN
					eRFID[ir4].nCardNumber			:=	P00_ReadRFIDCard.nReadedCardAfterScrewer;	
					bNewRFIDSaved					:=	TRUE;
					EXIT;
			 END_IF
		END_FOR	
		IF NOT bNewRFIDSaved THEN
			FOR ir4 := 1 TO 100 DO
				 IF eRFID[ir4].nCardNumber = 0 THEN
					eRFID[ir4]						:=	eClearPackageState;
					eRFID[ir4].nCardNumber			:=	P00_ReadRFIDCard.nReadedCardAfterScrewer;
					eRFID[ir4].bFormPresent 		:=	TRUE;
					EXIT;
				 END_IF
			END_FOR	
		END_IF
		bNewRFIDSaved := FALSE;	
	END_IF	
END_IF


(******************************************)
(************CZUJNIK POD ROBOTEM***********)
//Jeżeli wykryło kartę 
//stare rtReadedCardRobotTransfer(CLK:=P00_ReadRFIDCard.bReadedCardBottleTransfer,Q=>);
fbrtReadedCardRobotTransfer	(bIn:=P00_ReadRFIDCard.bReadedCardBottleTransfer,	tFilterTimeOn:=T#50MS,	tFilterTimeOff:=T#0MS);	//opózniony o 50ms żeby już był wczytany RFID
rtReadedCardRobotTransfer	(CLK:=fbrtReadedCardRobotTransfer.bOut,				Q=>);
//Stare IF rtReadedCardRobotTransfer.Q THEN
IF rtReadedCardRobotTransfer.Q THEN	
	nr5:=nr5+1;
	eRobotPackageState[2].bFormPresent:=TRUE; // dodane do testów 20.06 jak cos to wykomentować
	IF eRobotPackageState[2].bFormPresent  THEN
		eRobotPackageState[2].nCardNumber:=P00_ReadRFIDCard.nReadedCardBottleTransfer;
		FOR ir5 := 1 TO 100 DO
			 IF eRFID[ir5].nCardNumber = P00_ReadRFIDCard.nReadedCardBottleTransfer THEN
					eRobotPackageState[2]:=eRFID[ir5];			
					bNewRFIDSaved := TRUE;
			END_IF
		END_FOR	
		
		IF NOT bNewRFIDSaved THEN
			FOR ir5 := 1 TO 100 DO
				 IF eRFID[ir5].nCardNumber = 0 THEN
						eRFID[ir5] := eClearPackageState;
						eRFID[ir5].nCardNumber := P00_ReadRFIDCard.nReadedCardBottleTransfer;
						eRFID[ir5].bFormPresent := TRUE;
						eRobotPackageState[2]:=eRFID[ir5];	
						EXIT;
				 END_IF
			END_FOR	
		END_IF
	bNewRFIDSaved := FALSE;	
	END_IF
END_IF
bNewRFIDSaved := FALSE;	


(********KONIEC CZUJNIK POD ROBOTEM********)
(******************************************)

(**SOROTWANIE TABLICY***) 

	(*	FOR i := 1 TO 99 DO
			IF  eRFID[i].nCardNumber < eRFID[i+1].nCardNumber THEN
				eRFIDTemp :=  eRFID[i];	
				eRFID[i] := eRFID[i+1];
				eRFID[i+1] := eRFIDTemp;
			END_IF
		END_FOR*)
	
(***KONIEC SORTOWANIA TABLICY***)
END_ACTION

ACTION a2RFIDWeightingForm:
(*
Nazwa:			aRFIDWeightingForm
Opis:			Przeważanie formatek z RFID
Wersja:			v0.1
Data:			2019-11-12
Autor:			DP
Urzadzenia:		
Konfiguracja:	
Info:
- program na działać jak jest włączona zmienna VIS.bWeighingForm, wtedy działa normalny cykl
- po skończeniu przeważania ustawić zmienną bWeighingFormDone co zatrzyma cykl (zmienna ta jest w presistantach)
- koniec przeważania narazie po 2minutach
- pobieranie wartości  z przeważania tylko jak w recepturze wybrana jest waga formatki na 0
AnRFIDCardNumberShow: ARRAY [1..100] OF ULINT;							// Tabela numerów formatek 
AnRFIDWeightShow: ARRAY [1..100] OF LREAL;								// Tabela wag formatek	
*)


rtWeighingForm(CLK:=VIS.bWeighingForm,Q=>);
IF rtWeighingForm.Q THEN
	bWeighingFormReset	:= TRUE;	
	bWeighingAutoTarePreset	:= TRUE;
	bWeighingFormDone := FALSE;
	bWeighingFormDoneDialog := FALSE;
END_IF

rtWeightingDone(CLK:=(P05_Weight.fbWeight1.bCycleDone AND P05_Weight.fbWeight2.bCycleDone AND P05_Weight.fbWeight3.bCycleDone AND P05_Weight.fbWeight4.bCycleDone) ,Q=>); // tutaj był błąd bo powinna być też 4 waga
rtWeightingDone2Phase(CLK:=(P05_Weight.fbWeight5.bCycleDone AND P05_Weight.fbWeight6.bCycleDone), Q=>);

IF bDosingTwoPhases THEN
	tWeightTime:=T#20S; //bylo 4 m
ELSE
	tWeightTime:=T#20S; //bylo 3m  //potemm bylo 2.40m
END_IF

IF VIS.bWeighingForm  THEN
	IF diRFIDWeightingFormNumber=0 THEN
		IF bDosingTwoPhases THEN
			diRFIDWeightingFormNumber:=P00_ReadRFIDCard.fbAfterDispencers2PhaseReader.diReadedCode;
			ELSE
			diRFIDWeightingFormNumber:=P00_ReadRFIDCard.fbAfterDispencersReader.diReadedCode;
		END_IF
	END_IF
	IF tonAfter1stweight.Q THEN
		IF bDosingTwoPhases THEN
			IF P00_ReadRFIDCard.fbAfterDispencers2PhaseReader.diReadedCode = diRFIDWeightingFormNumber THEN
				bWeightEnd:=TRUE;
			END_IF
		ELSE
			IF P00_ReadRFIDCard.fbAfterDispencersReader.diReadedCode = diRFIDWeightingFormNumber THEN
				bWeightEnd:=TRUE;
			END_IF
		END_IF
	END_IF
ELSE
	bWeightEnd:=FALSE;
	diRFIDWeightingFormNumber:=0;
END_IF
tonAfter1stweight(IN:=NOT(diRFIDWeightingFormNumber=0),PT:=T#10S);

tonWeighingForm(IN:=VIS.bWeighingForm AND bWeightEnd AND P00_PackML.fbPMLAuto.ePMLState = E_PMLState.ePMLState_EXECUTE,PT:=tWeightTime);
tonWeighingForm.ET;

// kiedy wyłączone dozowanie dwufazowe

IF VIS.bWeighingForm AND rtWeightingDone.Q AND NOT bDosingTwoPhases THEN		
		FOR i := 1 TO 100 DO
			IF eWeightPackageState[1].nCardNumber = VIS.AnRFIDCardNumberShow[i] THEN	
				VIS.AnRFIDWeightShow[i] := VIS.lrWeight1Measured; 
				bNewRFIDSaved1 := TRUE;
			
			ELSIF eWeightPackageState[2].nCardNumber = VIS.AnRFIDCardNumberShow[i] THEN
				VIS.AnRFIDWeightShow[i] := VIS.lrWeight2Measured; 
				bNewRFIDSaved2 := TRUE;
			
			ELSIF eWeightPackageState[3].nCardNumber = VIS.AnRFIDCardNumberShow[i] THEN
				VIS.AnRFIDWeightShow[i] := VIS.lrWeight3Measured; 
				bNewRFIDSaved3 := TRUE;
			
			ELSIF eWeightPackageState[4].nCardNumber = VIS.AnRFIDCardNumberShow[i] THEN
				VIS.AnRFIDWeightShow[i] := VIS.lrWeight4Measured; 
				bNewRFIDSaved4 := TRUE;				
			END_IF;
	
		END_FOR
		
		IF NOT bNewRFIDSaved1 THEN
				FOR i := 1 TO 100 DO
					 IF VIS.AnRFIDCardNumberShow[i] = 0 THEN
							VIS.AnRFIDCardNumberShow[i] := eWeightPackageState[1].nCardNumber;
							VIS.AnRFIDWeightShow[i] := VIS.lrWeight1Measured; 			
							EXIT;
					 END_IF
				END_FOR	
		END_IF
		IF NOT bNewRFIDSaved2 THEN
				FOR i := 1 TO 100 DO
					 IF VIS.AnRFIDCardNumberShow[i] = 0 THEN
							VIS.AnRFIDCardNumberShow[i] := eWeightPackageState[2].nCardNumber;
							VIS.AnRFIDWeightShow[i] := VIS.lrWeight2Measured; 			
							EXIT;
					 END_IF
				END_FOR	
		END_IF		


		IF NOT bNewRFIDSaved3 THEN
				FOR i := 1 TO 100 DO
					 IF VIS.AnRFIDCardNumberShow[i] = 0 THEN
							VIS.AnRFIDCardNumberShow[i] := eWeightPackageState[3].nCardNumber;
							VIS.AnRFIDWeightShow[i] := VIS.lrWeight3Measured; 			
							EXIT;
					 END_IF
				END_FOR	
		END_IF		


		IF NOT bNewRFIDSaved4 THEN
				FOR i := 1 TO 100 DO
					 IF VIS.AnRFIDCardNumberShow[i] = 0 THEN
							VIS.AnRFIDCardNumberShow[i] := eWeightPackageState[4].nCardNumber;
							VIS.AnRFIDWeightShow[i] := VIS.lrWeight4Measured; 			
							EXIT;
					 END_IF
				END_FOR	
		END_IF		
		
		
		bNewRFIDSaved1:=FALSE;
		bNewRFIDSaved2:=FALSE;
		bNewRFIDSaved3:=FALSE;
		bNewRFIDSaved4:=FALSE;
END_IF




//----------------------------------------------------------------------------------------------------------------
// kiedy włączone dozowanie dwufazowe
IF VIS.bWeighingForm AND rtWeightingDone2Phase.Q AND  bDosingTwoPhases THEN		
		FOR i := 1 TO 100 DO
			IF eWeightPackage2PhasePackageState[1].nCardNumber = VIS.AnRFIDCardNumberShow[i] THEN	
				VIS.AnRFIDWeightShow[i] := VIS.lrWeight5Measured; 
				bNewRFIDSaved1 := TRUE;
			
			ELSIF eWeightPackage2PhasePackageState[2].nCardNumber = VIS.AnRFIDCardNumberShow[i] THEN
				VIS.AnRFIDWeightShow[i] := VIS.lrWeight6Measured; 
				bNewRFIDSaved2 := TRUE;
				
			END_IF;
	
		END_FOR
		
		IF NOT bNewRFIDSaved1 THEN
				FOR i := 1 TO 100 DO
					 IF VIS.AnRFIDCardNumberShow[i] = 0 THEN
							VIS.AnRFIDCardNumberShow[i] := eWeightPackage2PhasePackageState[1].nCardNumber;
							VIS.AnRFIDWeightShow[i] := VIS.lrWeight5Measured; 			
							EXIT;
					 END_IF
				END_FOR	
		END_IF
		IF NOT bNewRFIDSaved2 THEN
				FOR i := 1 TO 100 DO
					 IF VIS.AnRFIDCardNumberShow[i] = 0 THEN
							VIS.AnRFIDCardNumberShow[i] := eWeightPackage2PhasePackageState[2].nCardNumber;
							VIS.AnRFIDWeightShow[i] := VIS.lrWeight6Measured; 			
							EXIT;
					 END_IF
				END_FOR	
		END_IF		

		
		bNewRFIDSaved1:=FALSE;
		bNewRFIDSaved2:=FALSE;
END_IF


//---------------------------------------------------------------------------------------------------------------------------


//Resetowanie przeważania
IF bWeighingFormReset THEN
	FOR i := 1 TO 100 DO
		VIS.AnRFIDCardNumberShow[i]:=0;
		VIS.AnRFIDWeightShow[i]:=0;
	END_FOR
	bWeighingFormReset := FALSE;
	bWeighingFormDone := FALSE;
	bWeighingFormDoneDialog := FALSE;
END_IF

//Wyłączanie przeważania
IF tonWeighingForm.Q THEN //Wyłączanie przeważania
	bWeighingFormDone := TRUE;
	IF  NOT P_Persistent.fbUPS_CU8130.stStatus.ePowerStatus=2 THEN
		VIS.bWritePersistent := TRUE;
	END_IF
	VIS.bWritePersistent:=TRUE;
	VIS.bWeighingForm:=FALSE;
END_IF
END_ACTION

ACTION a2RFIDWeightingFormChecking:
//Informacja o niepoprawnym przeważeniu 

FOR i := 1 TO 100 DO
	IF VIS.AnRFIDWeightShow[i] > 0 THEN		
		lrAnRFIDWeightShowAverage		:=	VIS.AnRFIDWeightShow[i] + lrAnRFIDWeightShowAverage;
		iAnRFIDWeightShowAverageCount	:=	iAnRFIDWeightShowAverageCount	+	1;		
	END_IF
END_FOR	
//Średnia
IF iAnRFIDWeightShowAverageCount	=	0	THEN	iAnRFIDWeightShowAverageCount:=1;	END_IF
lrAnRFIDWeightShowAverage		:=	lrAnRFIDWeightShowAverage/iAnRFIDWeightShowAverageCount;
iAnRFIDWeightShowAverageCount	:=	0;

//Info jeżeli któraś formatka jest zła
bRFIDWeightShowAverageError :=	FALSE;
FOR i := 1 TO 100 DO
	IF VIS.AnRFIDWeightShow[i] > 0 AND ABS(lrAnRFIDWeightShowAverage - VIS.AnRFIDWeightShow[i]) > 40 THEN		
		bRFIDWeightShowAverageError :=	TRUE;
		ii := i;
	END_IF
END_FOR
END_ACTION

ACTION aAntyError:
(*
Nazwa:			aAI
Opis:			
Wersja:			v0.1
Data:			2025-08-29
Autor:			DP
Urzadzenia:		
Konfiguracja:	
Zmiany:
-20250829 [DP] Za robotem zmiana od czujnika, przed doz szlaban, 1D czujnik za
Info:
-


*)

(*****************Przed dozownikami	*****************)
// 1A - Ustawianie 4 formatki
tonFourthFormBeforeDispencerCheck.IN:=	NOT bDosingTwoPhases AND NOT IbFourthFormCheckFormSensor AND P00_PackML.fbPMLAuto.ePMLState = E_PMLState.ePMLState_EXECUTE AND P01_Gates.QbGateBeforeDispencersActuator AND
										NOT tonFourthFormBeforeDispencerCheck.Q;				
tonFourthFormBeforeDispencerCheck.PT:=	T#5S;;										
tonFourthFormBeforeDispencerCheck();											
IF tonFourthFormBeforeDispencerCheck.Q THEN
	eBeforeDispencersPackageState[4].bFormPresent:=FALSE;
	iRepairFourthFormBeforeDispencerCounter	:=	iRepairFourthFormBeforeDispencerCounter	+	1;
END_IF;

// 1B (2faza) - Autonaprawa 2 formatki przed dozowikiem 34
tonFourhtFormBeforeDispencer34(IN:= bDosingTwoPhases AND NOT IbFourthFormCheckFormSensor AND P00_PackML.fbPMLAuto.ePMLState = E_PMLState.ePMLState_EXECUTE AND 
									eBeforeDispencer34PackageState2Phase[2].bFormPresent AND NOT tonFourhtFormBeforeDispencer34.Q, PT:=T#10S);								
rttonFourtFormBeforeDispencer34Repair(CLK:=tonFourhtFormBeforeDispencer34.Q, Q=>);
IF rttonFourtFormBeforeDispencer34Repair.Q THEN
	eBeforeDispencer34PackageState2Phase[2].bFormPresent:=FALSE;
	iRepairBeforeDispencer34Counter:=iRepairBeforeDispencer34Counter+1;
END_IF

// 1C (2faza) - Autonaprawa jak jest butelka a niewydozowało
tonDispencer34DosingAborted( IN:= ((eDispencer34PackageState2Phase[1].bBottlePresent AND
							 (NOT eDispencer34PackageState2Phase[1].bDoseAborted OR NOT eDispencer34PackageState2Phase[1].bDosed)) OR
									(eDispencer34PackageState2Phase[2].bBottlePresent AND
							 (NOT eDispencer34PackageState2Phase[2].bDoseAborted OR  NOT eDispencer34PackageState2Phase[2].bDosed)))
							  AND (P00_PackML.fbPMLAuto.ePMLState = E_PMLState.ePMLState_EXECUTE) AND IbFourthFormCheckFormSensor , PT:=T#15S, ET=>); 

rttonDispencer34DosingAborted(CLK:=tonDispencer34DosingAborted.Q);
tonDispencer34DosingAborted.ET;				
IF rttonDispencer34DosingAborted.Q THEN
	IF (eDispencer34PackageState2Phase[1].bBottlePresent AND
		(NOT eDispencer34PackageState2Phase[1].bDoseAborted OR  NOT eDispencer34PackageState2Phase[1].bDosed))	THEN		
			eDispencer34PackageState2Phase[1].bDoseAborted:=TRUE;
			eDispencer34PackageState2Phase[1].bDosed:=FALSE;		
	END_IF
		
	IF (eDispencer34PackageState2Phase[2].bBottlePresent AND
		(NOT eDispencer34PackageState2Phase[2].bDoseAborted OR  NOT eDispencer34PackageState2Phase[2].bDosed))	THEN	
			eDispencer34PackageState2Phase[2].bDoseAborted:=TRUE;
			eDispencer34PackageState2Phase[2].bDosed:=FALSE;	
	END_IF	
	iCounterDispencer34DosingAborted:=	iCounterDispencer34DosingAborted+1;	
END_IF

// 1D - Ustawianie jak nie ma dwufazy // Ustawianie 1 2 3 4 formatki
tonFormBeforeDispenscerCheck.IN:=	IbFourthFormCheckFormSensor AND P00_PackML.fbPMLAuto.ePMLState = E_PMLState.ePMLState_EXECUTE AND NOT tonFormBeforeDispenscerCheck.Q
									AND NOT bDosingTwoPhases AND NOT P00_PackML.fbIbDispencerAfterCheckFormSensor.bOut;
tonFormBeforeDispenscerCheck.PT:=	T#10S; //bylo 15
tonFormBeforeDispenscerCheck();	

IF tonFormBeforeDispenscerCheck.Q THEN
	eBeforeDispencersPackageState[4].bFormPresent	:=	TRUE;
	eBeforeDispencersPackageState[3].bFormPresent	:=	TRUE;
	eBeforeDispencersPackageState[2].bFormPresent	:=	TRUE;
	eBeforeDispencersPackageState[1].bFormPresent	:=	TRUE;
	
	eDispencersPackageState[1].bFormPresent			:=	TRUE;
	eDispencersPackageState[2].bFormPresent			:=	TRUE;
	eDispencersPackageState[3].bFormPresent			:=	TRUE;
	eDispencersPackageState[4].bFormPresent			:=	TRUE;
	
	// Dodane na testy żeby nie sypało błędami RFID	
	IF 	eBeforeDispencersPackageState[4].nCardNumber =0 THEN	eBeforeDispencersPackageState[4].nCardNumber :=	999;	END_IF
	IF 	eBeforeDispencersPackageState[3].nCardNumber =0 THEN	eBeforeDispencersPackageState[3].nCardNumber :=	999;	END_IF
	IF 	eBeforeDispencersPackageState[2].nCardNumber =0 THEN	eBeforeDispencersPackageState[2].nCardNumber :=	999;	END_IF
	IF 	eBeforeDispencersPackageState[1].nCardNumber =0 THEN	eBeforeDispencersPackageState[1].nCardNumber :=	999;	END_IF	
	iRepairFormBeforeDispenscerCounter	:=	iRepairFormBeforeDispenscerCounter	+	1;	
END_IF

// 1E (2faza) - ustawianie jak jest dwufaza - Ustawianie 1 2  formatki
tonFormBeforeDispenscer2PhaseCheck.IN:=	IbFourthFormCheckFormSensor AND P00_PackML.fbPMLAuto.ePMLState = E_PMLState.ePMLState_EXECUTE AND NOT tonFormBeforeDispenscer2PhaseCheck.Q
									AND bDosingTwoPhases AND 
									(NOT eBeforeDispencer34PackageState2Phase[1].bFormPresent OR NOT eBeforeDispencer34PackageState2Phase[1].bFormPresent)
									;
tonFormBeforeDispenscer2PhaseCheck.PT:=	T#5S;
tonFormBeforeDispenscer2PhaseCheck();	

IF tonFormBeforeDispenscer2PhaseCheck.Q THEN
	eBeforeDispencer34PackageState2Phase[1].bFormPresent	:=	TRUE;
	eBeforeDispencer34PackageState2Phase[2].bFormPresent	:=	TRUE;
	
	//dodane żeby nie sypało błędami	
	IF eBeforeDispencer34PackageState2Phase[1].nCardNumber=0 THEN		eBeforeDispencer34PackageState2Phase[1].nCardNumber:=999;	END_IF
	IF eBeforeDispencer34PackageState2Phase[2].nCardNumber=0 THEN		eBeforeDispencer34PackageState2Phase[2].nCardNumber:=999;	END_IF
	iRepairFormBeforeDispenscer2PhaseCounter	:=	iRepairFormBeforeDispenscer2PhaseCounter	+	1;
END_IF

(*****************Pod dozownikami	*****************)
//DoseAborted v2
tonDispencerRepair1 (IN:=
					P00_PackML.iDispencersCase = 3 AND
					P00_PackML.fbPMLAuto.ePMLState = E_PMLState.ePMLState_EXECUTE AND P00_PackML.bDispencersReady AND P00_PackML.bCatchersready AND
					NOT P02_Dispencers.fbDispencer1.bCycleDone	AND
					NOT P02_Dispencers.fbDispencer2.bCycleDone 	AND
					NOT P02_Dispencers.fbDispencer3.bCycleDone 	AND
					NOT P02_Dispencers.fbDispencer4.bCycleDone 	AND
					(
						(eDispencersPackageState[1].bDosed OR eDispencersPackageState[1].bDoseAborted) OR
						(eDispencersPackageState[2].bDosed OR eDispencersPackageState[2].bDoseAborted) OR 
						(eDispencersPackageState[3].bDosed OR eDispencersPackageState[3].bDoseAborted) OR 
						(eDispencersPackageState[4].bDosed OR eDispencersPackageState[4].bDoseAborted) 
					) AND
					(
					(NOT eDispencersPackageState[1].bDosed AND NOT eDispencersPackageState[1].bDoseAborted) OR
					(NOT eDispencersPackageState[2].bDosed AND NOT eDispencersPackageState[2].bDoseAborted) OR
					(NOT eDispencersPackageState[3].bDosed AND NOT eDispencersPackageState[3].bDoseAborted) OR 
					(NOT eDispencersPackageState[4].bDosed AND NOT eDispencersPackageState[4].bDoseAborted) 
					) AND				
				 	NOT tonDispencerRepair1.Q,
					PT:=T#15S);
					tonDispencerRepair1.ET;
IF tonDispencerRepair1.Q THEN
					iDispencerRepair1	:=	iDispencerRepair1	+	1;
					eDispencersPackageState[1].bDosed	:=	eDispencersPackageState[1].bDoseAborted	:=	TRUE;
					eDispencersPackageState[2].bDosed	:=	eDispencersPackageState[2].bDoseAborted :=	TRUE;
					eDispencersPackageState[3].bDosed	:=	eDispencersPackageState[3].bDoseAborted :=	TRUE;
					eDispencersPackageState[4].bDosed	:=	eDispencersPackageState[4].bDoseAborted	:=	TRUE;
END_IF


(******************Autonaprawa za dozownikami*************************)
// 1 - Kasowanie rejestrow jezeli nie ma nic na czujnikach 
tonAfterDispencersRepair(IN:=NOT P05_Weight.tonIbWeight1FormSensor.Q AND NOT P05_Weight.tonIbWeight2FormSensor.Q  AND NOT P05_Weight.tonIbWeight3FormSensor.Q  AND NOT P05_Weight.tonIbWeight4FormSensor.Q  AND
						NOT P00_ReadRFIDCard.bReadedCardAfterDispencers AND 
						(
						eAfterDispencersPackageState[4].bFormPresent OR
						eAfterDispencersPackageState[3].bFormPresent OR
						eAfterDispencersPackageState[2].bFormPresent OR
						eAfterDispencersPackageState[1].bFormPresent OR
						eWeightPackageState[4].bFormPresent			OR
						eWeightPackageState[3].bFormPresent 		OR
						eWeightPackageState[2].bFormPresent			OR
						eWeightPackageState[1].bFormPresent				
						) AND (P00_PackML.fbPMLAuto.ePMLState = E_PMLState.ePMLState_EXECUTE) AND
						NOT
						P01_Gates.QbGateBeforeWeight14Actuator AND 
						NOT MAIN.IbTwoPhasesFormSensorBetweenDispencers AND 
						NOT tonAfterDispencersRepair.Q
, PT:=T#10S); //bylo 15


IF tonAfterDispencersRepair.Q THEN
	FOR ia:=1 TO 4 DO	
		//eAfterDispencersPackageState[ia].bFormPresent:=FALSE;
		eWeightPackageState[iw].bFormPresent		:=FALSE;	
	END_FOR
	itonAfterDispencersRepair		:=itonAfterDispencersRepair+1;
END_IF

tonAfterDispencersRepair1B(IN:=NOT P02_Dispencers.IbDispencerAfterCheckFormSensor AND 	
						NOT P00_ReadRFIDCard.bReadedCardAfterDispencers	
						 AND (P00_PackML.fbPMLAuto.ePMLState = E_PMLState.ePMLState_EXECUTE) AND
						NOT
						P01_Gates.QbGateBeforeWeight14Actuator AND 
						NOT MAIN.IbTwoPhasesFormSensorBetweenDispencers AND 
						NOT tonAfterDispencersRepair1B.Q 
						AND (eAfterDispencersPackageState[4].bFormPresent OR
						eAfterDispencersPackageState[3].bFormPresent OR
						eAfterDispencersPackageState[2].bFormPresent OR
						eAfterDispencersPackageState[1].bFormPresent)
, PT:=T#10S); //bylo 15


IF tonAfterDispencersRepair1B.Q THEN
	FOR ia:=1 TO 4 DO	
		eAfterDispencersPackageState[ia].bFormPresent:=FALSE;
		eWeightPackageState[iw].bFormPresent		:=FALSE;	
	END_FOR
	itonAfterDispencersRepair1B		:=itonAfterDispencersRepair1B+1;
END_IF



// 1 - Koniec ------------------------------------------------------------

// 2 - Kasowanie rejestrow jezeli nei ma nic na czujnikach----------------
tonAfterDispencersRepair2(IN:=NOT P05_Weight.tonIbWeight1FormSensor.Q AND NOT P05_Weight.tonIbWeight2FormSensor.Q AND NOT P05_Weight.tonIbWeight3FormSensor.Q AND NOT P05_Weight.tonIbWeight4FormSensor.Q AND
						NOT P00_ReadRFIDCard.bReadedCardAfterDispencers AND 
						(
						eWeightPackageState[4].bFormPresent			OR
						eWeightPackageState[3].bFormPresent 		OR
						eWeightPackageState[2].bFormPresent			OR
						eWeightPackageState[1].bFormPresent				
						) AND (P00_PackML.fbPMLAuto.ePMLState = E_PMLState.ePMLState_EXECUTE) AND
						P01_Gates.QbGateBeforeWeight14Actuator
, PT:=T#15S);

IF tonAfterDispencersRepair2.Q THEN
	FOR iw:=1 TO 4 DO	
		eWeightPackageState[iw].bFormPresent		:=FALSE;
	END_FOR
	itonAfterDispencersRepair2		:=itonAfterDispencersRepair2+1;
END_IF
// 2 - Koniec -----------------------------------------------------------

// 3 - Kasowanie rejestrow jezeli nei ma nic na czujnikach --------------
tonAfterDispencersRepair3(IN:=NOT P05_Weight.tonIbWeight1FormSensor.Q AND NOT P05_Weight.tonIbWeight2FormSensor.Q AND NOT P05_Weight.tonIbWeight3FormSensor.Q AND NOT P05_Weight.tonIbWeight4FormSensor.Q AND
						NOT P00_ReadRFIDCard.bReadedCardAfterDispencers AND 
						(
						eAfterDispencersPackageState[4].bFormPresent OR
						eAfterDispencersPackageState[3].bFormPresent OR
						eAfterDispencersPackageState[2].bFormPresent OR
						eAfterDispencersPackageState[1].bFormPresent OR
						eWeightPackageState[4].bFormPresent			OR
						eWeightPackageState[3].bFormPresent 		OR
						eWeightPackageState[2].bFormPresent			OR
						eWeightPackageState[1].bFormPresent				
						) AND (P00_PackML.fbPMLAuto.ePMLState = E_PMLState.ePMLState_EXECUTE) AND						
						P01_Gates.QbGateBeforeWeight14Actuator AND 
						NOT MAIN.IbTwoPhasesFormSensorBetweenDispencers AND NOT
						tonAfterDispencersRepair3.Q					
, PT:=T#8S);//bylo 15

IF tonAfterDispencersRepair3.Q THEN
	FOR ia:=4 TO 1 BY -1 DO	
		IF eAfterDispencersPackageState[ia].bFormPresent THEN
			;//eAfterDispencersPackageState[ia].bFormPresent:=FALSE;
			EXIT;
		END_IF
	END_FOR
	itonAfterDispencersRepair3		:=itonAfterDispencersRepair3+1;
END_IF
// 3 - Koniec ------------------------------------------------------------

// 4- Kasowanie rejestrow jezeli nei ma nic na czujnikach-------------
(*iAfterDispencersFormCounter := 	BOOL_TO_INT(eAfterDispencersPackageState[4].bFormPresent) +
								BOOL_TO_INT(eAfterDispencersPackageState[3].bFormPresent) +
								BOOL_TO_INT(eAfterDispencersPackageState[2].bFormPresent) +
								BOOL_TO_INT(eAfterDispencersPackageState[1].bFormPresent);

tonAfterDispencersRepair4(IN:=
								(iAfterDispencersFormCounter >= 1 AND iAfterDispencersFormCounter < 4) AND 
								P00_PackML.fbPMLAuto.ePMLState = E_PMLState.ePMLState_EXECUTE AND						
								P01_Gates.QbGateBeforeWeight14Actuator AND 
								NOT tonAfterDispencersRepair4.Q				
, PT:=T#20S);
IF tonAfterDispencersRepair4.Q THEN
	FOR ia:=4 TO 1 BY -1 DO	
		eAfterDispencersPackageState[ia].bFormPresent:=TRUE;
	END_FOR
	itonAfterDispencersRepair4		:=itonAfterDispencersRepair4+1;
END_IF*)
// 4 - Koniec ------------------------------------------------------------


// 4 - (2faza) Kssowanie za 1 i 2 dozownikiem jak dwufaza -----------------------
tonAfterDispencer12Repair( IN:= NOT P05_Weight.IbWeight6FormSensor AND NOT P05_Weight.IbWeight5FormSensor AND NOT MAIN.IbSecondFormCheckFormSensor AND
								(eAfterDispencer12PackageState2Phase[1].bFormPresent OR eAfterDispencer12PackageState2Phase[2].bFormPresent
								 OR eWeightPackage2PhasePackageState[1].bFormPresent OR eWeightPackage2PhasePackageState[2].bFormPresent )
								AND ((P00_PackML.fbPMLAuto.ePMLState = E_PMLState.ePMLState_EXECUTE) OR (P00_PackML.fbPMLAuto.ePMLState = E_PMLState.ePMLState_STOPPING)) AND 
								NOT tonAfterDispencer12Repair.Q, PT:=T#20S);	
rttonAfterDispencer12Repair(CLK:=tonAfterDispencer12Repair.Q);
						
IF rttonAfterDispencer12Repair.Q THEN
	eAfterDispencer12PackageState2Phase[1]:=eClearPackageState;
	eAfterDispencer12PackageState2Phase[2]:=eClearPackageState;
	eWeightPackage2PhasePackageState[1]:=eClearPackageState;
	eWeightPackage2PhasePackageState[2]:=eClearPackageState;
	GVL.iRepairAfterDispencerCounter:=GVL.iRepairAfterDispencerCounter+1;
	
END_IF;
// 4 - Koniec ----------------------------------------------------------

// 5 - (2faza) Dodawanie formatek przed 12 jak stoją za 34 ---------------------
tonAfterDispencer1234Repair(IN:= bDosingTwoPhases AND
								Main.IbTwoPhasesFormSensorBetweenDispencers  AND bFormTransportersScrewerCmdStart AND
								(NOT eBeforeDispencer12PackageState2Phase[1].bFormPresent OR NOT eBeforeDispencer12PackageState2Phase[2].bFormPresent OR
								NOT eDispencer12PackageState2Phase[1].bFormPresent OR NOT eDispencer12PackageState2Phase[2].bFormPresent
								) AND  
								((P00_PackML.fbPMLAuto.ePMLState = E_PMLState.ePMLState_EXECUTE) OR (P00_PackML.fbPMLAuto.ePMLState = E_PMLState.ePMLState_STOPPING)) AND
								NOT tonAfterDispencer1234Repair.Q
								 , PT:=T#6S);
								 
rttonAfterDispencer1234Repair(CLK:=tonAfterDispencer1234Repair.Q,Q=>);

IF rttonAfterDispencer1234Repair.Q THEN	
	eDispencer12PackageState2Phase[1].bFormPresent			:=	TRUE;	
	eDispencer12PackageState2Phase[2].bFormPresent			:=	TRUE;
	eDispencer34PackageState2Phase[1].bFormPresent			:=	TRUE;	
	eDispencer34PackageState2Phase[2].bFormPresent			:=	TRUE;		
	eBeforeDispencer12PackageState2Phase[1].bFormPresent	:=	TRUE;
	eBeforeDispencer12PackageState2Phase[2].bFormPresent	:=	TRUE;
	iRepairBeforeDispencer12Counter:=iRepairBeforeDispencer12Counter+1;
END_IF
// 5 - Koniec ----------------------------------------------------------

// 5B - (2faza) Usuwanie formatek przed 12 ---------------------
tonAfterDispencer1234Repair2	(IN:= bDosingTwoPhases AND
								NOT Main.IbTwoPhasesFormSensorBetweenDispencers  AND bFormTransportersScrewerCmdStart AND
								(eBeforeDispencer12PackageState2Phase[1].bFormPresent OR eBeforeDispencer12PackageState2Phase[2].bFormPresent OR 
								eAfterDispencer34PackageState2Phase[1].bFormPresent OR eAfterDispencer34PackageState2Phase[2].bFormPresent
								) AND  
								((P00_PackML.fbPMLAuto.ePMLState = E_PMLState.ePMLState_EXECUTE) OR (P00_PackML.fbPMLAuto.ePMLState = E_PMLState.ePMLState_STOPPING)) AND
								NOT tonAfterDispencer1234Repair2.Q
								 , PT:=T#6S);						

IF tonAfterDispencer1234Repair2.Q THEN	
	eAfterDispencer34PackageState2Phase[1].bFormPresent		:=	FALSE;
	eAfterDispencer34PackageState2Phase[2].bFormPresent		:=	FALSE;
	eBeforeDispencer12PackageState2Phase[1].bFormPresent	:=	FALSE;
	eBeforeDispencer12PackageState2Phase[2].bFormPresent	:=	FALSE;
	iRepairBeforeDispencer12Counter2:=iRepairBeforeDispencer12Counter2+1;
END_IF
// 5B - Koniec ----------------------------------------------------------







//6 - kasowanie ( zdarza się przy wyłączeniu i włączeniu wag*)
tonWeightRepair1( IN:= P05_Weight.fbWeightStation.eRunningState=E_WeightLiftStationState.eRepair AND
							(eWeightPackageState[1].bFormPresent OR eWeightPackageState[2].bFormPresent OR eWeightPackageState[3].bFormPresent OR eWeightPackageState[4].bFormPresent) AND 
							((P00_PackML.fbPMLAuto.ePMLState = E_PMLState.ePMLState_EXECUTE) OR (P00_PackML.fbPMLAuto.ePMLState = E_PMLState.ePMLState_STOPPING)) AND 
							NOT tonWeightRepair1.Q, PT:=T#6S);	

IF tonWeightRepair1.Q THEN
	eWeightPackageState[1].bFormPresent := FALSE;
	eWeightPackageState[2].bFormPresent := FALSE;
	eWeightPackageState[3].bFormPresent := FALSE;
	eWeightPackageState[4].bFormPresent := FALSE;
	iWeightRepair1Counter	:=	iWeightRepair1Counter	+	1;
END_IF
// 6 - Koniec ----------------------------------------------------------

//7 - kasowanie ( zdarza się ze waga 0*)
tonWeightRepair2( IN:= VIS.lrDispencer1WeightMeasured = 0 AND VIS.lrDispencer2WeightMeasured = 0 AND VIS.lrDispencer3WeightMeasured = 0 AND VIS.lrDispencer4WeightMeasured = 0 AND
						(eWeightPackageState[1].bFormPresent) AND bWeight1Enable AND
						(P00_PackML.fbPMLAuto.ePMLState = E_PMLState.ePMLState_EXECUTE) AND 
						NOT tonWeightRepair2.Q, PT:=T#6S);	

IF tonWeightRepair2.Q THEN
	eWeightPackageState[1].bFormPresent 	:= FALSE;
	iWeightRepair2Counter					:=	iWeightRepair2Counter	+	1;
END_IF
// 6 - Koniec ----------------------------------------------------------



(*****Autonaprawa pod sorterem nasadek**********)
// 1A- Ustawianie 1 2 3 4 formatki
tonFormBeforeCapSorterCheck.IN:=	P00_PackML.fbIbCapSorterFourthFormCheckFormSensor.bOut AND P00_PackML.fbPMLAuto.ePMLState = E_PMLState.ePMLState_EXECUTE AND NOT tonFormBeforeCapSorterCheck.Q AND
									
										(	NOT eBeforeCapSorterPackageState[4].bFormPresent OR
											NOT eBeforeCapSorterPackageState[3].bFormPresent OR	
											NOT eBeforeCapSorterPackageState[2].bFormPresent OR
											NOT eBeforeCapSorterPackageState[1].bFormPresent 										
										)

 									AND 
									bFormTransportersScrewerCmdStart
									;
tonFormBeforeCapSorterCheck.PT:=	T#5S;
tonFormBeforeCapSorterCheck();	

IF tonFormBeforeCapSorterCheck.Q THEN
	eBeforeCapSorterPackageState[4].bFormPresent	:=	TRUE;
	eBeforeCapSorterPackageState[3].bFormPresent	:=	TRUE;
	eBeforeCapSorterPackageState[2].bFormPresent	:=	TRUE;
	eBeforeCapSorterPackageState[1].bFormPresent	:=	TRUE;
	
	eCapSorterPackageState[1].bFormPresent			:=	TRUE;
	eCapSorterPackageState[2].bFormPresent			:=	TRUE;
	eCapSorterPackageState[3].bFormPresent			:=	TRUE;
	eCapSorterPackageState[4].bFormPresent			:=	TRUE;
	
	// Dodane na testy żeby nie sypało błędami RFID	
	IF 	eBeforeCapSorterPackageState[4].nCardNumber =0 THEN		eBeforeCapSorterPackageState[4].nCardNumber :=	999;END_IF
	IF 	eBeforeCapSorterPackageState[3].nCardNumber =0 THEN		eBeforeCapSorterPackageState[3].nCardNumber :=	999;END_IF
	IF 	eBeforeCapSorterPackageState[2].nCardNumber =0 THEN		eBeforeCapSorterPackageState[2].nCardNumber :=	999;END_IF
	IF 	eBeforeCapSorterPackageState[1].nCardNumber =0 THEN		eBeforeCapSorterPackageState[1].nCardNumber :=	999;END_IF
	itonFormBeforeCapSorterCheck	:=	itonFormBeforeCapSorterCheck	+	1;
END_IF
// 1A - Koniec


(*****Autonaprawa przed zakręcarkami*********)
(*...*)
	

(****** Autonaprawa pod zakręcarkami*********)
// 1A - 
tonUnderScrewerFormStuck1(IN:= (eUnderScrewerPackageState[1].bCapGripperScrewed OR eUnderScrewerPackageState[1].bCapGripperScrewAborted
								OR eUnderScrewerPackageState[2].bCapGripperScrewed OR eUnderScrewerPackageState[2].bCapGripperScrewAborted ) 
								AND NOT eAfterScrewerPackageState[1].bFormPresent AND NOT eAfterScrewerPackageState[2].bFormPresent 
								AND P09_CapPuttedCheck.IbCapPuttedCheckFormSensor AND P10_GripperScrewer.IbGripperScrewersThirdFormCheckFormSensor
								 AND (P00_PackML.fbPMLAuto.ePMLState = E_PMLState.ePMLState_EXECUTE), PT:=T#12S);
rttonUnderScrewerFormStuck1(CLK:=tonUnderScrewerFormStuck1.Q);
							
	
IF rttonUnderScrewerFormStuck1.Q THEN		
		IF (NOT eUnderScrewerPackageState[2].bCapGripperScrewed) THEN
			eUnderScrewerPackageState[2].bCapGripperScrewAborted :=TRUE;
		END_IF

		IF (NOT eUnderScrewerPackageState[1].bCapGripperScrewed) THEN
			eUnderScrewerPackageState[1].bCapGripperScrewAborted :=TRUE;
		END_IF
	
	iScrewerFormStuck:=iScrewerFormStuck+1;
END_IF

// 1B -  jak nie odczytra RFID
tonUnderScrewerFormStuck2(IN:= 	(NOT eBeforeScrewers2PackageState[2].bFormPresent OR
								NOT eBeforeScrewers2PackageState[1].bFormPresent OR
								NOT eBeforeScrewersPackageState[2].bFormPresent OR
								NOT eBeforeScrewersPackageState[1].bFormPresent) AND
								P00_PackML.iScrewerDragCase=10 AND
								P00_PackML.tonThirdFormsSensor.Q AND
								P00_PackML.tonAfterScreweEmpty.Q AND
								P00_PackML.fbIbCapSorterGateScrewerSensor.bOUT		
								AND (P00_PackML.fbPMLAuto.ePMLState = E_PMLState.ePMLState_EXECUTE)
								AND NOT tonUnderScrewerFormStuck2.Q
								,PT:=T#25S);
IF tonUnderScrewerFormStuck2.Q THEN		
	eBeforeScrewers2PackageState[2].bFormPresent	:=	TRUE;
	eBeforeScrewers2PackageState[1].bFormPresent	:=	TRUE;
	eBeforeScrewersPackageState[2].bFormPresent		:=	TRUE;
	eBeforeScrewersPackageState[1].bFormPresent		:=	TRUE;
	iScrewerFormStuck2:=iScrewerFormStuck2+1;
END_IF
(****** Autonaprawa za zakręcarkami*********)
// 1A - 
tonAfterScrewerFormStuck1(IN:= 	(eAfterScrewerPackageState[1].bFormPresent OR
								eAfterScrewerPackageState[2].bFormPresent) AND
								NOT P11_CapCorrectCheck.IbCapCorrectCheckAfterScrewerFormSensor AND
								NOT P11_CapCorrectCheck.IbCapCorrectCheckDialAfterScrewerFormSensor	
								AND (P00_PackML.fbPMLAuto.ePMLState = E_PMLState.ePMLState_EXECUTE)
								AND NOT tonAfterScrewerFormStuck1.Q
								,PT:=T#8S);
IF tonAfterScrewerFormStuck1.Q THEN		
	eAfterScrewerPackageState[1].bFormPresent	:=	FALSE;
	eAfterScrewerPackageState[2].bFormPresent	:=	FALSE;
	iScrewerFormStuck3:=iScrewerFormStuck3+1;
END_IF
		
(*****Autonaprawa pod robotem**********)
//Jak jest przeniesiona na etykieciarke
tonRobotPackageStatebBottleTransferedToLabeler	(IN:=(eRobotPackageState[1].bBottleTransferedToLabeler OR eRobotPackageState[1].bBottleTransferedToExit) AND NOT P00_PackML.fbIbBottleTransferFormAfterSensor.bOut,	PT:=T#10S);
tonRobotPackageStatebBottleTransferedToLabeler2	(IN:=(eRobotPackageState[2].bBottleTransferedToLabeler OR eRobotPackageState[2].bBottleTransferedToExit) AND NOT P00_PackML.fbIbBottleTransferFormAfterSensor.bOut,	PT:=T#10S);

//Naprawa jak sa za długo dwie formatki
tonRobotPackageState1FormsTooLong	(IN:=P13_BottleTransfer.IbFirstFormCheckFormSensor AND NOT eRobotPackageState[1].bFormPresent, PT:=T#10S);
tonRobotPackageState2FormsTooLong	(IN:=P13_BottleTransfer.IbSecondFormCheckFormSensor AND NOT eRobotPackageState[2].bFormPresent, PT:=T#10S);

rttonRobotPackageState1FormsTooLong	(CLK:=tonRobotPackageState1FormsTooLong.Q);
rttonRobotPackageState2FormsTooLong	(CLK:=tonRobotPackageState2FormsTooLong.Q);

IF rttonRobotPackageState1FormsTooLong.Q THEN
	eRobotPackageState[1].bFormPresent:=TRUE;
	IF 	eRobotPackageState[1].nCardNumber=0 THEN
		eRobotPackageState[1].nCardNumber:=999; 
		eRobotPackageState[1].bBottlePresent:=TRUE;
		eRobotPackageState[1].bCapGripperScrewed:=FALSE;
	END_IF
	iRobotRepairPackageForm1Counter:= iRobotRepairPackageForm1Counter+1;
END_IF

IF rttonRobotPackageState2FormsTooLong.Q THEN
	eRobotPackageState[2].bFormPresent:=TRUE;
	IF 	eRobotPackageState[2].nCardNumber=0 THEN 
		eRobotPackageState[2].nCardNumber:=P00_ReadRFIDCard.nReadedCardBottleTransfer;
	END_IF
	iRobotRepairPackageForm2Counter:= iRobotRepairPackageForm2Counter+1;	
END_IF

rttonRobotPackageStatebBottleTransferedToLabeler	(CLK:=	tonRobotPackageStatebBottleTransferedToLabeler.Q);
rttonRobotPackageStatebBottleTransferedToLabeler2	(CLK:=	tonRobotPackageStatebBottleTransferedToLabeler2.Q);

//Jak utknie pierwsza formatka
IF rttonRobotPackageStatebBottleTransferedToLabeler.Q THEN
	eRobotPackageState[1].bBottleTransferedToLabeler 	:= FALSE;
	eRobotPackageState[1].bBottleTransferedToExit 		:= FALSE;
	itonRobotBottleTransferedToLabelerRepair			:= 	itonRobotBottleTransferedToLabelerRepair	+	1;
END_IF

//Jak utknie druga formatka					
IF  rttonRobotPackageStatebBottleTransferedToLabeler2.Q THEN
	eRobotPackageState[2].bBottleTransferedToLabeler 	:= FALSE;
	eRobotPackageState[2].bBottleTransferedToExit 		:= FALSE;
	itonRobotBottleTransferedToLabeler2Repair			:= 	itonRobotBottleTransferedToLabeler2Repair	+	1;
END_IF
	
rteUnderScrewerPackageStateCheck	(CLK:=	eUnderScrewerPackageState[1].bCapGripperScrewAborted);
rteUnderScrewerPackageStateCheck2	(CLK:=	eUnderScrewerPackageState[2].bCapGripperScrewAborted);

IF rteUnderScrewerPackageStateCheck.Q THEN
	iUnderScrewerPackageStateCheckCounter :=iUnderScrewerPackageStateCheckCounter+1;
END_IF

IF rteUnderScrewerPackageStateCheck2.Q THEN
	iUnderScrewerPackageStateCheckCounter2 :=iUnderScrewerPackageStateCheckCounter2+1;
END_IF



(*Kasowanie*)
IF bResetAntyErrorCounters THEN
	bResetAntyErrorCounters	:=	FALSE;
	// 1A - Ustawianie 4 formatki
	iRepairFourthFormBeforeDispencerCounter	:=	0;
	// 1B (2faza) - Autonaprawa 2 formatki przed dozowikiem 34
	iRepairBeforeDispencer34Counter	:=	0;
	// 1C (2faza) - Autonaprawa jak jest butelka a niewydozowało
	iCounterDispencer34DosingAborted	:=	0;
	// 1D - Ustawianie jak nie ma dwufazy // Ustawianie 1 2 3 4 formatki
	iRepairFormBeforeDispenscerCounter	:=	0;										//10s
	// 1E (2faza) - ustawianie jak jest dwufaza - Ustawianie 1 2  formatki
	iRepairFormBeforeDispenscer2PhaseCounter	:=	0;
	(******************Pod dozownikami*************************)	
	// 1 - DoseAborted v2
	iDispencerRepair1:=	0;
	(******************Za dozownikami*************************)
	// 1 - Kasowanie rejestrow jezeli nie ma nic na czujnikach 
	itonAfterDispencersRepair	:=	0;												//10s
	// 2 - Kasowanie rejestrow jezeli nei ma nic na czujnikach----------------
	itonAfterDispencersRepair2	:=	0;
	// 3 - Kasowanie rejestrow jezeli nei ma nic na czujnikach --------------
	itonAfterDispencersRepair3	:=	0;
	// 4- Kasowanie rejestrow jezeli nei ma nic na czujnikach-------------
	itonAfterDispencersRepair4	:=	0;
	// 4 - (2faza) Kssowanie za 1 i 2 dozownikiem jak dwufaza -----------------------
	iRepairAfterDispencerCounter	:=	0;
	// 5 - (2faza) Dodawanie formatek przed 12 jak stoją za 34 ---------------------
	iRepairBeforeDispencer12Counter	:=	0;
	// 5B - (2faza) Usuwanie formatek przed 12  ---------------------	
	iRepairBeforeDispencer12Counter2 := 0;
	// 6 - kasowanie rej przy wył. i wł wag
	iWeightRepair1Counter := 0;
	// 7 - kasowanie rej gdy waga 0
	iWeightRepair2Counter := 0;	
	(*****Autonaprawa pod sorterem nasadek**********)
	// 1A- Ustawianie 1 2 3 4 formatki
	itonFormBeforeCapSorterCheck	:=	0;
	(****** Autonaprawa pod zakręcarkami*********)
	// 1A - 
	iScrewerFormStuck	:=	0;
	// 1B - Jezeli nie odczyta RFID 
	iScrewerFormStuck2	:=	0;
	(****** Autonaprawa za zakręcarkami*********)	
	iScrewerFormStuck3	:=	0;
	(*****Autonaprawa pod robotem**********)
	//Jak jest przeniesiona na etykieciarke
	iRobotRepairPackageForm1Counter	:=	0;
	iRobotRepairPackageForm2Counter	:=	0;
	//Jak utknie pierwsza formatka
	itonRobotBottleTransferedToLabelerRepair	:=	0;
	//Jak utknie druga formatka	
	itonRobotBottleTransferedToLabeler2Repair	:=	0;

END_IF
END_ACTION

ACTION aAntyErrorLidFeeder:
IbLidFeederThirdFormSensor 	;
IbLidFeederAfterSensor ;		
IbLidSealerSecondFormSensor ;
IbLidSealerAfterSensor 	;	

IF bLidFeederEnable OR bWickFeederEnable THEN
	
(*****************Autonaprawa 1 LidFeeder*****************)
// 1 - Przed pojadnikiem platynek
	tonRepairLidFeeder1		(	IN	:=	IbLidFeederThirdFormSensor AND 
										( 
											//NOT eBeforeLidFeeder2PackageState[1].bFormPresent OR //dp
											NOT eBeforeLidFeederPackageState[2].bFormPresent OR
											NOT eBeforeLidFeederPackageState[1].bFormPresent 
										) AND
										P00_PackML.fbPMLAuto.ePMLState = E_PMLState.ePMLState_EXECUTE AND NOT tonRepairLidFeeder1.Q,
								PT	:=	T#5S
							);																
									
	IF tonRepairLidFeeder1.Q THEN
		//eBeforeLidFeeder2PackageState[1].bFormPresent	:=	TRUE;	
		eBeforeLidFeederPackageState[2].bFormPresent	:=	TRUE;	//dp	
		eBeforeLidFeederPackageState[1].bFormPresent	:=	TRUE;	//dp	
		iRepairLidFeeder1Counter						:=	iRepairLidFeeder1Counter	+	1;
	END_IF;

(*****************Autonaprawa 2 LidFeeder*****************)
// 2 - Przed zgrzewaniem platynek
	tonRepairLidFeeder2		(	IN	:=	IbLidSealerFirstFormSensor AND NOT IbLidSealerSecondFormSensor AND
										( 										
											NOT eBeforeLidSealerPackageState[1].bFormPresent 
										) AND
										P00_PackML.fbPMLAuto.ePMLState = E_PMLState.ePMLState_EXECUTE AND NOT tonRepairLidFeeder2.Q,
								PT	:=	T#5S
							);																
									
	IF tonRepairLidFeeder2.Q THEN	
		eBeforeLidSealerPackageState[1].bFormPresent	:=	TRUE;		
		iRepairLidFeeder2Counter						:=	iRepairLidFeeder2Counter	+	1;
	END_IF;
	
// 3 - Przed zgrzewaniem platynek	
	tonRepairLidFeeder3		(	IN	:=	IbLidSealerFirstFormSensor AND IbLidSealerSecondFormSensor AND 
										(
										( 										
											NOT eBeforeLidSealerPackageState[1].bFormPresent AND 
											eBeforeLidSealerPackageState[2].bFormPresent 
										) OR
										( 										
											eBeforeLidSealerPackageState[1].bFormPresent AND 
											NOT eBeforeLidSealerPackageState[2].bFormPresent 
										) OR
										( 										
											NOT eBeforeLidSealerPackageState[1].bFormPresent AND 
											NOT eBeforeLidSealerPackageState[2].bFormPresent 
										)												
										)
 										AND
										P00_PackML.fbPMLAuto.ePMLState = E_PMLState.ePMLState_EXECUTE AND NOT tonRepairLidFeeder3.Q,
								PT	:=	T#5S
							);																
									
	IF tonRepairLidFeeder3.Q THEN
		eBeforeLidSealerPackageState[2].bFormPresent	:=	TRUE;		
		eBeforeLidSealerPackageState[1].bFormPresent	:=	TRUE;		
		iRepairLidFeeder3Counter						:=	iRepairLidFeeder3Counter	+	1;
	END_IF;
	
(*****************Autonaprawa 3 LidFeeder*****************)
// 4 - Przed zgrzewaniem platynek
		tonRepairLidFeeder4		(	IN	:=	NOT IbLidFeederAfterSensor AND 
										( 										
											eAfterLidFeederPackageState[2].bFormPresent OR
											eAfterLidFeederPackageState[1].bFormPresent 										
										) AND
										P00_PackML.fbPMLAuto.ePMLState = E_PMLState.ePMLState_EXECUTE AND NOT tonRepairLidFeeder4.Q,
								PT	:=	T#8S
							);																
									
	IF tonRepairLidFeeder4.Q THEN
		eAfterLidFeederPackageState[2].bFormPresent		:=	FALSE;		
		eAfterLidFeederPackageState[1].bFormPresent		:=	FALSE;		
		iRepairLidFeeder4Counter						:=	iRepairLidFeeder4Counter	+	1;
	END_IF;
		
	
	
END_IF
END_ACTION

ACTION aAntyErrorROPP:
(*
P07_ROPP.IbROPPSevenFormSensor;	
P07_ROPP.IbROPPThirdFormSensor;	
P07_ROPP.IbROPPAfterFormSensor;	
P07_ROPP.IbROPPAfter2FormSensor	;

IF bROPPCappingEnable THEN
	
(*****************Autonaprawa 1 ROPP*****************)
// 1 - Przed 
	tonRepairROPP1		(	IN	:=	IbLidFeederThirdFormSensor AND 
										( 
											NOT eBeforeLidFeeder2PackageState[1].bFormPresent OR
											NOT eBeforeLidFeederPackageState[2].bFormPresent OR
											NOT eBeforeLidFeederPackageState[1].bFormPresent 
										) AND
										P00_PackML.fbPMLAuto.ePMLState = E_PMLState.ePMLState_EXECUTE AND NOT tonRepairROPP1.Q,
								PT	:=	T#5S
							);																
									
	IF tonRepairROPP1.Q THEN
		//eBeforeLidFeeder2PackageState[1].bFormPresent	:=	TRUE;	
		//eBeforeLidFeederPackageState[2].bFormPresent	:=	TRUE;		
		//eBeforeLidFeederPackageState[1].bFormPresent	:=	TRUE;		
		iRepairROPP1Counter								:=	iRepairROPP1Counter	+	1;
	END_IF;

(*****************Autonaprawa 2 ROPP*****************)
// 2 - Przed 
	tonRepairROPP2		(	IN	:=	IbLidSealerSecondFormSensor AND 
										( 										
											NOT eBeforeLidSealerPackageState[2].bFormPresent OR
											NOT eBeforeLidSealerPackageState[1].bFormPresent 
										) AND
										P00_PackML.fbPMLAuto.ePMLState = E_PMLState.ePMLState_EXECUTE AND NOT tonRepairROPP2.Q,
								PT	:=	T#5S
							);																
									
	IF tonRepairROPP2.Q THEN
		//eBeforeLidSealerPackageState[2].bFormPresent	:=	TRUE;		
		//eBeforeLidSealerPackageState[1].bFormPresent	:=	TRUE;		
		iRepairROPP2Counter								:=	iRepairROPP2Counter	+	1;
	END_IF;

(*****************Autonaprawa 3 ROPP*****************)
// 3 - Przed 
	tonRepairROPP3		(	IN	:=	NOT IbLidSealerSecondFormSensor AND 
										( 										
											eAfterLidFeederPackageState[2].bFormPresent OR
											eAfterLidFeederPackageState[1].bFormPresent OR 
											eBeforeLidSealerPackageState[2].bFormPresent
										) AND
										P00_PackML.fbPMLAuto.ePMLState = E_PMLState.ePMLState_EXECUTE AND NOT tonRepairROPP3.Q,
								PT	:=	T#8S
							);																
									
	IF tonRepairROPP3.Q THEN
		//eAfterLidFeederPackageState[2].bFormPresent		:=	FALSE;		
		//eAfterLidFeederPackageState[1].bFormPresent		:=	FALSE;		
		//eBeforeLidSealerPackageState[2].bFormPresent	:=	FALSE;		
		iRepairROPP3Counter								:=	iRepairROPP3Counter	+	1;
	END_IF;
	
(*****************Autonaprawa 4 ROPP*****************)
// 4 - 
	tonRepairROPP4		(	IN	:=	NOT IbLidSealerSecondFormSensor AND 
										( 										
											eAfterLidFeederPackageState[2].bFormPresent OR
											eAfterLidFeederPackageState[1].bFormPresent OR 
											eBeforeLidSealerPackageState[2].bFormPresent
										) AND
										P00_PackML.fbPMLAuto.ePMLState = E_PMLState.ePMLState_EXECUTE AND NOT tonRepairROPP4.Q,
								PT	:=	T#8S
							);																
									
	IF tonRepairROPP4.Q THEN
		//eAfterLidFeederPackageState[2].bFormPresent	:=	FALSE;		
		//eAfterLidFeederPackageState[1].bFormPresent	:=	FALSE;		
		//eBeforeLidSealerPackageState[2].bFormPresent	:=	FALSE;		
		iRepairROPP4Counter								:=	iRepairROPP4Counter	+	1;
	END_IF;	
	
END_IF
*)
END_ACTION

ACTION aBadPackage:


fb2ReasonBadPackageWithID(
						bEnable:=TRUE, 
						tTime:= T#24H,  
                        bReason1			:= 	(
												(NOT eRobotPackageState[1].bWeightTooLow AND NOT eRobotPackageState[1].bWeightTooHigh AND NOT eRobotPackageState[1].bWeightOK) OR  
												 NOT eRobotPackageState[1].bDosed
												 )
												AND 
												eRobotPackageState[1].bBottlePresent,
                        sReason1Description	:= '11',//'Brak dozy',//'DB',						
                        bReason2			:= eRobotPackageState[1].bWeightTooLow 			AND eRobotPackageState[1].bBottlePresent,
                        sReason2Description	:= '12',//'Waga za mała',//'WZM',
                        bReason3			:= eRobotPackageState[1].bWeightTooHigh 		AND eRobotPackageState[1].bBottlePresent,
                        sReason3Description	:= '13',//'Waga za duża', //było WZD
						bReason4			:= NOT eRobotPackageState[1].bLidPutted AND eRobotPackageState[1].bBottlePresent AND bLidFeederEnable,
						sReason4Description	:= '14', //było BOP
						bReason5			:= NOT eRobotPackageState[1].bLidPuttedOK AND eRobotPackageState[1].bBottlePresent AND bLidPuttedCheckEnable,
						sReason5Description	:= '15 ', //było PZO
						bReason6			:= NOT eRobotPackageState[1].bLidSealed AND eRobotPackageState[1].bBottlePresent AND bLidSealerEnable,
						sReason6Description	:= '16', //było BNZS
                        bReason7			:= NOT eRobotPackageState[1].bROPPPutted 		AND eRobotPackageState[1].bBottlePresent AND bROPPCappingEnable,
                        sReason7Description:= '22',//'ROPP nie nałożony',
                        bReason8			:= NOT eRobotPackageState[1].bROPPCapped 		AND eRobotPackageState[1].bBottlePresent AND bROPPCappingEnable,
                        sReason8Description:= '23',//'ROPP nie zakręcony',
                        bReason9			:= NOT eRobotPackageState[1].bROPPCappingOK 	AND eRobotPackageState[1].bBottlePresent AND bROPPCappingEnable,
                        sReason9Description:= '24',//'ROPP brak za stacją'																										
						bReason10			:= eRobotPackageState[1].bCapSorterPutted AND eRobotPackageState[1].bCapSorterPuttedAborted AND eRobotPackageState[1].bBottlePresent AND stCapSorterRead.bEnable AND NOT bCapSorterDisable,
						sReason10Description	:= '17', //było BNZS
                        bReason11			:= NOT eRobotPackageState[1].bCapOK 			AND eRobotPackageState[1].bBottlePresent,
                        sReason11Description	:= '18',//'Brak nasadki przed zakr.',//'BNPZ-Przed zak.1',
                        bReason12			:= NOT eRobotPackageState[1].bCapGripperScrewed AND eRobotPackageState[1].bBottlePresent,
                        sReason12Description	:= '19',//'Niezakręcona zakr.',//'NZZSZ',
                        bReason13			:= NOT eRobotPackageState[1].bCapCorrectCapOn 	AND eRobotPackageState[1].bBottlePresent,
                        sReason13Description:= '20',//'Brak nasadki za zakr.',//'BNZZ',
                        bReason14			:= eRobotPackageState[1].bCapCorrectNOK 		AND eRobotPackageState[1].bBottlePresent,
                        sReason14Description:= '21',//'Nasadka źle zakręcona',//'NZZ',
                        
						bReason21			:= (
												(NOT eRobotPackageState[2].bWeightTooLow AND NOT eRobotPackageState[2].bWeightTooHigh AND NOT eRobotPackageState[2].bWeightOK) OR
												NOT eRobotPackageState[2].bDosed
												)
												AND 
												eRobotPackageState[2].bBottlePresent,
                        sReason21Description	:= '11',//'Brak dozy',//'DB',			
                        bReason22			:= eRobotPackageState[2].bWeightTooLow 			AND eRobotPackageState[2].bBottlePresent,
                        sReason22Description	:= '12',//'Waga za mała',//'WZM',
                        bReason23			:= eRobotPackageState[2].bWeightTooHigh 		AND eRobotPackageState[2].bBottlePresent,
                        sReason23Description	:= '13',//'Waga za duża', //było WZD
						bReason24			:= NOT eRobotPackageState[2].bLidPutted AND eRobotPackageState[2].bBottlePresent AND bLidFeederEnable,
						sReason24Description	:= '14', //było BOP
						bReason25			:= NOT eRobotPackageState[2].bLidPuttedOK AND eRobotPackageState[2].bBottlePresent AND bLidPuttedCheckEnable,
						sReason25Description	:= '15', //było PZO
						bReason26			:= NOT eRobotPackageState[2].bLidSealed AND eRobotPackageState[2].bBottlePresent AND bLidSealerEnable,
						sReason26Description	:= '16', //było BNZS
                     	bReason27			:= NOT eRobotPackageState[2].bROPPPutted 		AND eRobotPackageState[2].bBottlePresent AND bROPPCappingEnable,
                        sReason27Description:= '22',//'ROPP nie nałożony',
                        bReason28			:= NOT eRobotPackageState[2].bROPPCapped 		AND eRobotPackageState[2].bBottlePresent AND bROPPCappingEnable,
                        sReason28Description:= '23',//'ROPP nie zakręcony',
                        bReason29			:= NOT eRobotPackageState[2].bROPPCappingOK 	AND eRobotPackageState[2].bBottlePresent AND bROPPCappingEnable,
                        sReason29Description:= '24',//'ROPP brak za stacją'																							
						bReason210			:= eRobotPackageState[2].bCapSorterPutted 		AND eRobotPackageState[2].bCapSorterPuttedAborted AND eRobotPackageState[2].bBottlePresent AND stCapSorterRead.bEnable AND NOT bCapSorterDisable,
						sReason210Description	:= '17', //było BNZS								
                        bReason211			:= NOT eRobotPackageState[2].bCapOK 			AND eRobotPackageState[2].bBottlePresent,
                        sReason211Description	:= '18',//'Brak nasadki przed zakr.',//'BNPZ-Przed zak.1',
                        bReason212			:= NOT eRobotPackageState[2].bCapGripperScrewed AND eRobotPackageState[2].bBottlePresent,
                        sReason212Description	:= '19',//'Niezakręcona zakr.',//'NZZSZ',
                        bReason213			:= NOT eRobotPackageState[2].bCapCorrectCapOn 	AND eRobotPackageState[2].bBottlePresent,
                        sReason213Description:= '20',//'Brak nasadki za zakr.',//'BNZZ',
                        bReason214			:= eRobotPackageState[2].bCapCorrectNOK 		AND eRobotPackageState[2].bBottlePresent,
                        sReason214Description:= '21',//'Nasadka źle zakręcona',//'NZZ',


						AStReason=> VIS.AStBadPackageReason, 
						bClear:=VIS.bBadPackageReasonReset,
						bAddReason1:= bAddBadPackageReason, 
						bAddReason2:= bAddBadPackageReason2						
						);	
			
						
						VIS.sBadPackageReason1	:= WSTRING_TO_STRING((WConcat(UDINT_TO_WSTRING(VIS.AStBadPackageReason[0].udiID),VIS.AStBadPackageReason[0].wsDescription)));
		                VIS.sBadPackageReason2	:= WSTRING_TO_STRING((WConcat(UDINT_TO_WSTRING(VIS.AStBadPackageReason[1].udiID),VIS.AStBadPackageReason[1].wsDescription)));
                        VIS.sBadPackageReason3	:= WSTRING_TO_STRING((WConcat(UDINT_TO_WSTRING(VIS.AStBadPackageReason[2].udiID),VIS.AStBadPackageReason[2].wsDescription)));
END_ACTION

ACTION aBadPackage_1:
(*	

fbReasonBadPackage1(
						bEnable:=TRUE, 
						bReset:= , 
						tTime:= T#10M,  
						bAddReason:= bAddBadPackageReason, 
                        bReason1			:= 	(
												//(NOT eRobotPackageState[1].bWeightTooLow AND NOT eRobotPackageState[1].bWeightTooHigh AND NOT eRobotPackageState[1].bWeightOK) OR 
												 eRobotPackageState[1].bDoseAborted
												 )
												AND 
												eRobotPackageState[1].bBottlePresent,
                        sReason1Description	:= 'Empty',//'Brak dozy',//'DB',						
                        bReason2			:= eRobotPackageState[1].bWeightTooLow 			AND eRobotPackageState[1].bBottlePresent,
                        sReason2Description	:= 'Weight too low',//'Waga za mała',//'WZM',
                        bReason3			:= eRobotPackageState[1].bWeightTooHigh 		AND eRobotPackageState[1].bBottlePresent,
                        sReason3Description	:= 'Weight too high',//'Waga za duża', //było WZD
						bReason4			:= NOT eRobotPackageState[1].bLidPutted AND eRobotPackageState[1].bBottlePresent AND bLidFeederEnable,
						sReason4Description	:= 'Brak odłożenia platynki', //było BOP
						bReason5			:= NOT eRobotPackageState[1].bLidPuttedOK AND eRobotPackageState[1].bBottlePresent AND bLidPuttedCheckEnable,
						sReason5Description	:= 'Platynka źle odłożona ', //było PZO
						bReason6			:= NOT eRobotPackageState[1].bLidSealed AND eRobotPackageState[1].bBottlePresent AND bLidSealerEnable,
						sReason6Description	:= 'Platynka nie zgrzana', //było BNZS
						bReason7			:= eRobotPackageState[1].bCapSorterPutted AND eRobotPackageState[1].bCapSorterPuttedAborted AND eRobotPackageState[1].bBottlePresent AND stCapSorterRead.bEnable AND NOT bCapSorterDisable,
						sReason7Description	:= 'Brak nas.(słomka) ', //było BNZS
                        bReason8			:= NOT eRobotPackageState[1].bCapOK 			AND eRobotPackageState[1].bBottlePresent,
                        sReason8Description	:= 'No cap before capper',//'Brak nasadki przed zakr.',//'BNPZ-Przed zak.1',
                        bReason9			:= NOT eRobotPackageState[1].bCapGripperScrewed AND eRobotPackageState[1].bBottlePresent,
                        sReason9Description	:= 'Wrong capping',//'Niezakręcona zakr.',//'NZZSZ',
                        bReason10			:= NOT eRobotPackageState[1].bCapCorrectCapOn 	AND eRobotPackageState[1].bBottlePresent,
                        sReason10Description:= 'No cap after capping',//'Brak nasadki za zakr.',//'BNZZ',
                        bReason11			:= eRobotPackageState[1].bCapCorrectNOK 		AND eRobotPackageState[1].bBottlePresent,
                        sReason11Description:= 'Cap not screwed (after cap.)',//'Nasadka źle zakręcona',//'NZZ',
                        bReason12			:= ,
                        sReason12Description:= , 
						sBadPackage1=> sBadPackage1Reason1, 
						sBadPackage2=> sBadPackage1Reason2, 
						sBadPackage3=> sBadPackage1Reason3,
						iBadPackage1=> iBadPackage1ReasonCount1, 
						iBadPackage2=> iBadPackage1ReasonCount2, 
						iBadPackage3=> iBadPackage1ReasonCount3, 
						);	
			
	fbReasonBadPackage2(
						bEnable:= TRUE, 
						bReset:= , 
						tTime:= T#10M,  
						//bAddReason:= bAddBadPackageReason AND P00_PackML.nCounterFormsToLoad=2,
						bAddReason:= bAddBadPackageReason,// AND P00_PackML.nCounterFormsToLoad=2,
						
                        bReason1			:= (
												//(NOT eRobotPackageState[2].bWeightTooLow AND NOT eRobotPackageState[2].bWeightTooHigh AND NOT eRobotPackageState[2].bWeightOK) OR
												eRobotPackageState[2].bDoseAborted
												)
												AND 
												eRobotPackageState[2].bBottlePresent,
                        sReason1Description	:= 'Empty',//'Brak dozy',//'DB',			
                        bReason2			:= eRobotPackageState[2].bWeightTooLow 			AND eRobotPackageState[2].bBottlePresent,
                        sReason2Description	:= 'Weight too low',//'Waga za mała',//'WZM',
                        bReason3			:= eRobotPackageState[2].bWeightTooHigh 		AND eRobotPackageState[2].bBottlePresent,
                        sReason3Description	:= 'Weight too high',//'Waga za duża', //było WZD
						bReason4			:= NOT eRobotPackageState[2].bLidPutted AND eRobotPackageState[2].bBottlePresent AND bLidFeederEnable,
						sReason4Description	:= 'Brak odłożenia platynki', //było BOP
						bReason5			:= NOT eRobotPackageState[2].bLidPuttedOK AND eRobotPackageState[2].bBottlePresent AND bLidPuttedCheckEnable,
						sReason5Description	:= 'Platynka źle odłożona ', //było PZO
						bReason6			:= NOT eRobotPackageState[2].bLidSealed AND eRobotPackageState[2].bBottlePresent AND bLidSealerEnable,
						sReason6Description	:= 'Platynka nie zgrzana', //było BNZS
						bReason7			:= eRobotPackageState[2].bCapSorterPutted 		AND eRobotPackageState[2].bCapSorterPuttedAborted AND eRobotPackageState[2].bBottlePresent AND stCapSorterRead.bEnable AND NOT bCapSorterDisable,
						sReason7Description	:= 'Brak nas.(słomka)', //było BNZS								
                        bReason8			:= NOT eRobotPackageState[2].bCapOK 			AND eRobotPackageState[2].bBottlePresent,
                        sReason8Description	:= 'No cap before capper',//'Brak nasadki przed zakr.',//'BNPZ-Przed zak.1',
                        bReason9			:= NOT eRobotPackageState[2].bCapGripperScrewed AND eRobotPackageState[2].bBottlePresent,
                        sReason9Description	:= 'Wrong capping',//'Niezakręcona zakr.',//'NZZSZ',
                        bReason10			:= NOT eRobotPackageState[2].bCapCorrectCapOn 	AND eRobotPackageState[2].bBottlePresent,
                        sReason10Description:= 'No cap after capping',//'Brak nasadki za zakr.',//'BNZZ',
                        bReason11			:= eRobotPackageState[2].bCapCorrectNOK 		AND eRobotPackageState[2].bBottlePresent,
                        sReason11Description:= 'Cap not screwed (after cap.)',//'Nasadka źle zakręcona',//'NZZ',
                        bReason12			:= ,
                        sReason12Description	:= , 
						sBadPackage1=> sBadPackage2Reason1, 
						sBadPackage2=> sBadPackage2Reason2, 
						sBadPackage3=> sBadPackage2Reason3,
						iBadPackage1=> iBadPackage2ReasonCount1, 
						iBadPackage2=> iBadPackage2ReasonCount2, 
						iBadPackage3=> iBadPackage2ReasonCount3,
						);
						
		//VIS.sBadPackageReason1 			:=	CONCAT(CONCAT(sBadPackage1Reason1,';'),sBadPackage2Reason1);
		//VIS.sBadPackageReason2 			:=	CONCAT(CONCAT(sBadPackage1Reason2,';'),sBadPackage2Reason2);
		//VIS.sBadPackageReason3 			:=	CONCAT(CONCAT(sBadPackage1Reason3,';'),sBadPackage2Reason3);
		//VIS.iBadPackageReasonCount1			:=	iBadPackage1ReasonCount1 +	iBadPackage2ReasonCount1;
		//VIS.iBadPackageReasonCount2			:=	iBadPackage1ReasonCount2 +	iBadPackage2ReasonCount2;
		//VIS.iBadPackageReasonCount3			:=	iBadPackage1ReasonCount3 +	iBadPackage2ReasonCount3;		
		
